LIN {X -167.693,Y -83.818,Z 210.000,A 0.000,B 0.000,C 180.000,E1 0.000} C_DIS
LIN {X -163.156,Y -92.341,Z 210.000,A 0.000,B 0.000,C 180.000,E1 0.000} C_DIS
LIN {X -158.186,Y -100.617,Z 210.000,A 0.000,B 0.000,C 180.000,E1 0.000} C_DIS
LIN {X -152.797,Y -108.627,Z 210.000,A 0.000,B 0.000,C 180.000,E1 0.000} C_DIS
LIN {X -147.002,Y -116.348,Z 210.000,A 0.000,B 0.000,C 180.000,E1 0.000} C_DIS
LIN {X -140.817,Y -123.762,Z 210.000,A 0.000,B 0.000,C 180.000,E1 0.000} C_DIS
LIN {X -134.260,Y -130.847,Z 210.000,A 0.000,B 0.000,C 180.000,E1 0.000} C_DIS
LIN {X -127.346,Y -137.585,Z 210.000,A 0.000,B 0.000,C 180.000,E1 0.000} C_DIS
LIN {X -120.095,Y -143.957,Z 210.000,A 0.000,B 0.000,C 180.000,E1 0.000} C_DIS
LIN {X -112.524,Y -149.949,Z 210.000,A 0.000,B 0.000,C 180.000,E1 0.000} C_DIS
LIN {X -104.656,Y -155.543,Z 210.000,A 0.000,B 0.000,C 180.000,E1 0.000} C_DIS
LIN {X -96.510,Y -160.725,Z 210.000,A 0.000,B 0.000,C 180.000,E1 0.000} C_DIS
LIN {X -88.108,Y -165.480,Z 210.000,A 0.000,B 0.000,C 180.000,E1 0.000} C_DIS
LIN {X -79.474,Y -169.796,Z 210.000,A 0.000,B 0.000,C 180.000,E1 0.000} C_DIS
LIN {X -70.624,Y -173.663,Z 210.000,A 0.000,B 0.000,C 180.000,E1 0.000} C_DIS
LIN {X -61.594,Y -177.067,Z 210.000,A 0.000,B 0.000,C 180.000,E1 0.000} C_DIS
LIN {X -52.397,Y -180.003,Z 210.000,A 0.000,B 0.000,C 180.000,E1 0.000} C_DIS
LIN {X -43.061,Y -182.462,Z 210.000,A 0.000,B 0.000,C 180.000,E1 0.000} C_DIS
LIN {X -33.610,Y -184.437,Z 210.000,A 0.000,B 0.000,C 180.000,E1 0.000} C_DIS
LIN {X -24.072,Y -185.923,Z 210.000,A 0.000,B 0.000,C 180.000,E1 0.000} C_DIS
LIN {X -14.469,Y -186.915,Z 210.000,A 0.000,B 0.000,C 180.000,E1 0.000} C_DIS
LIN {X -4.827,Y -187.412,Z 210.000,A 0.000,B 0.000,C 180.000,E1 0.000} C_DIS
LIN {X 4.827,Y -187.412,Z 210.000,A 0.000,B 0.000,C 180.000,E1 0.000} C_DIS
LIN {X 14.469,Y -186.915,Z 210.000,A 0.000,B 0.000,C 180.000,E1 0.000} C_DIS
LIN {X 24.072,Y -185.923,Z 210.000,A 0.000,B 0.000,C 180.000,E1 0.000} C_DIS
LIN {X 33.610,Y -184.437,Z 210.000,A 0.000,B 0.000,C 180.000,E1 0.000} C_DIS
LIN {X 43.061,Y -182.462,Z 210.000,A 0.000,B 0.000,C 180.000,E1 0.000} C_DIS
LIN {X 52.397,Y -180.003,Z 210.000,A 0.000,B 0.000,C 180.000,E1 0.000} C_DIS
LIN {X 61.593,Y -177.068,Z 210.000,A 0.000,B 0.000,C 180.000,E1 0.000} C_DIS
LIN {X 70.627,Y -173.662,Z 210.000,A 0.000,B 0.000,C 180.000,E1 0.000} C_DIS
LIN {X 79.474,Y -169.796,Z 210.000,A 0.000,B 0.000,C 180.000,E1 0.000} C_DIS
LIN {X 88.108,Y -165.480,Z 210.000,A 0.000,B 0.000,C 180.000,E1 0.000} C_DIS
LIN {X 96.510,Y -160.725,Z 210.000,A 0.000,B 0.000,C 180.000,E1 0.000} C_DIS
LIN {X 104.656,Y -155.543,Z 210.000,A 0.000,B 0.000,C 180.000,E1 0.000} C_DIS
LIN {X 112.524,Y -149.949,Z 210.000,A 0.000,B 0.000,C 180.000,E1 0.000} C_DIS
LIN {X 120.095,Y -143.957,Z 210.000,A 0.000,B 0.000,C 180.000,E1 0.000} C_DIS
LIN {X 127.346,Y -137.585,Z 210.000,A 0.000,B 0.000,C 180.000,E1 0.000} C_DIS
LIN {X 134.261,Y -130.846,Z 210.000,A 0.000,B 0.000,C 180.000,E1 0.000} C_DIS
LIN {X 140.817,Y -123.762,Z 210.000,A 0.000,B 0.000,C 180.000,E1 0.000} C_DIS
LIN {X 147.002,Y -116.348,Z 210.000,A 0.000,B 0.000,C 180.000,E1 0.000} C_DIS
LIN {X 152.797,Y -108.627,Z 210.000,A 0.000,B 0.000,C 180.000,E1 0.000} C_DIS
LIN {X 158.186,Y -100.617,Z 210.000,A 0.000,B 0.000,C 180.000,E1 0.000} C_DIS
LIN {X 163.156,Y -92.341,Z 210.000,A 0.000,B 0.000,C 180.000,E1 0.000} C_DIS
LIN {X 167.693,Y -83.818,Z 210.000,A 0.000,B 0.000,C 180.000,E1 0.000} C_DIS
LIN {X 171.786,Y -75.075,Z 210.000,A 0.000,B 0.000,C 180.000,E1 0.000} C_DIS
LIN {X 175.422,Y -66.133,Z 210.000,A 0.000,B 0.000,C 180.000,E1 0.000} C_DIS
LIN {X 178.595,Y -57.013,Z 210.000,A 0.000,B 0.000,C 180.000,E1 0.000} C_DIS
LIN {X 181.293,Y -47.744,Z 210.000,A 0.000,B 0.000,C 180.000,E1 0.000} C_DIS
LIN {X 183.511,Y -38.347,Z 210.000,A 0.000,B 0.000,C 180.000,E1 0.000} C_DIS
LIN {X 185.241,Y -28.852,Z 210.000,A 0.000,B 0.000,C 180.000,E1 0.000} C_DIS
LIN {X 186.480,Y -19.276,Z 210.000,A 0.000,B 0.000,C 180.000,E1 0.000} C_DIS
LIN {X 187.226,Y -9.650,Z 210.000,A 0.000,B 0.000,C 180.000,E1 0.000} C_DIS
LIN {X 187.474,Y 0.000,Z 210.000,A 0.000,B 0.000,C 180.000,E1 0.000} C_DIS
LIN {X 187.226,Y 9.650,Z 210.000,A 0.000,B 0.000,C 180.000,E1 0.000} C_DIS
LIN {X 186.480,Y 19.276,Z 210.000,A 0.000,B 0.000,C 180.000,E1 0.000} C_DIS
LIN {X 185.241,Y 28.852,Z 210.000,A 0.000,B 0.000,C 180.000,E1 0.000} C_DIS
LIN {X 183.511,Y 38.347,Z 210.000,A 0.000,B 0.000,C 180.000,E1 0.000} C_DIS
LIN {X 181.293,Y 47.744,Z 210.000,A 0.000,B 0.000,C 180.000,E1 0.000} C_DIS
LIN {X 178.595,Y 57.013,Z 210.000,A 0.000,B 0.000,C 180.000,E1 0.000} C_DIS
LIN {X 175.422,Y 66.133,Z 210.000,A 0.000,B 0.000,C 180.000,E1 0.000} C_DIS
LIN {X 171.786,Y 75.075,Z 210.000,A 0.000,B 0.000,C 180.000,E1 0.000} C_DIS
LIN {X 167.693,Y 83.818,Z 210.000,A 0.000,B 0.000,C 180.000,E1 0.000} C_DIS
LIN {X 163.156,Y 92.341,Z 210.000,A 0.000,B 0.000,C 180.000,E1 0.000} C_DIS
LIN {X 158.186,Y 100.617,Z 210.000,A 0.000,B 0.000,C 180.000,E1 0.000} C_DIS
LIN {X 152.797,Y 108.627,Z 210.000,A 0.000,B 0.000,C 180.000,E1 0.000} C_DIS
LIN {X 147.002,Y 116.348,Z 210.000,A 0.000,B 0.000,C 180.000,E1 0.000} C_DIS
LIN {X 140.817,Y 123.762,Z 210.000,A 0.000,B 0.000,C 180.000,E1 0.000} C_DIS
LIN {X 134.260,Y 130.847,Z 210.000,A 0.000,B 0.000,C 180.000,E1 0.000} C_DIS
LIN {X 127.346,Y 137.585,Z 210.000,A 0.000,B 0.000,C 180.000,E1 0.000} C_DIS
LIN {X 120.095,Y 143.957,Z 210.000,A 0.000,B 0.000,C 180.000,E1 0.000} C_DIS
LIN {X 112.524,Y 149.949,Z 210.000,A 0.000,B 0.000,C 180.000,E1 0.000} C_DIS
LIN {X 104.656,Y 155.543,Z 210.000,A 0.000,B 0.000,C 180.000,E1 0.000} C_DIS
LIN {X 96.510,Y 160.725,Z 210.000,A 0.000,B 0.000,C 180.000,E1 0.000} C_DIS
LIN {X 88.108,Y 165.480,Z 210.000,A 0.000,B 0.000,C 180.000,E1 0.000} C_DIS
LIN {X 79.474,Y 169.796,Z 210.000,A 0.000,B 0.000,C 180.000,E1 0.000} C_DIS
LIN {X 70.624,Y 173.663,Z 210.000,A 0.000,B 0.000,C 180.000,E1 0.000} C_DIS
LIN {X 61.594,Y 177.067,Z 210.000,A 0.000,B 0.000,C 180.000,E1 0.000} C_DIS
LIN {X 52.397,Y 180.003,Z 210.000,A 0.000,B 0.000,C 180.000,E1 0.000} C_DIS
LIN {X 43.061,Y 182.462,Z 210.000,A 0.000,B 0.000,C 180.000,E1 0.000} C_DIS
LIN {X 33.610,Y 184.437,Z 210.000,A 0.000,B 0.000,C 180.000,E1 0.000} C_DIS
LIN {X 24.072,Y 185.923,Z 210.000,A 0.000,B 0.000,C 180.000,E1 0.000} C_DIS
LIN {X 14.469,Y 186.915,Z 210.000,A 0.000,B 0.000,C 180.000,E1 0.000} C_DIS
LIN {X 4.827,Y 187.412,Z 210.000,A 0.000,B 0.000,C 180.000,E1 0.000} C_DIS
LIN {X -4.827,Y 187.412,Z 210.000,A 0.000,B 0.000,C 180.000,E1 0.000} C_DIS
LIN {X -14.469,Y 186.915,Z 210.000,A 0.000,B 0.000,C 180.000,E1 0.000} C_DIS
LIN {X -24.072,Y 185.923,Z 210.000,A 0.000,B 0.000,C 180.000,E1 0.000} C_DIS
LIN {X -33.610,Y 184.437,Z 210.000,A 0.000,B 0.000,C 180.000,E1 0.000} C_DIS
LIN {X -43.061,Y 182.462,Z 210.000,A 0.000,B 0.000,C 180.000,E1 0.000} C_DIS
LIN {X -52.397,Y 180.003,Z 210.000,A 0.000,B 0.000,C 180.000,E1 0.000} C_DIS
LIN {X -61.593,Y 177.068,Z 210.000,A 0.000,B 0.000,C 180.000,E1 0.000} C_DIS
LIN {X -70.627,Y 173.662,Z 210.000,A 0.000,B 0.000,C 180.000,E1 0.000} C_DIS
LIN {X -79.474,Y 169.796,Z 210.000,A 0.000,B 0.000,C 180.000,E1 0.000} C_DIS
LIN {X -88.108,Y 165.480,Z 210.000,A 0.000,B 0.000,C 180.000,E1 0.000} C_DIS
LIN {X -96.510,Y 160.725,Z 210.000,A 0.000,B 0.000,C 180.000,E1 0.000} C_DIS
LIN {X -104.656,Y 155.543,Z 210.000,A 0.000,B 0.000,C 180.000,E1 0.000} C_DIS
LIN {X -112.524,Y 149.949,Z 210.000,A 0.000,B 0.000,C 180.000,E1 0.000} C_DIS
LIN {X -120.095,Y 143.957,Z 210.000,A 0.000,B 0.000,C 180.000,E1 0.000} C_DIS
LIN {X -127.346,Y 137.585,Z 210.000,A 0.000,B 0.000,C 180.000,E1 0.000} C_DIS
LIN {X -134.261,Y 130.846,Z 210.000,A 0.000,B 0.000,C 180.000,E1 0.000} C_DIS
LIN {X -140.817,Y 123.762,Z 210.000,A 0.000,B 0.000,C 180.000,E1 0.000} C_DIS
LIN {X -147.002,Y 116.348,Z 210.000,A 0.000,B 0.000,C 180.000,E1 0.000} C_DIS
LIN {X -152.797,Y 108.627,Z 210.000,A 0.000,B 0.000,C 180.000,E1 0.000} C_DIS
LIN {X -158.186,Y 100.617,Z 210.000,A 0.000,B 0.000,C 180.000,E1 0.000} C_DIS
LIN {X -163.156,Y 92.341,Z 210.000,A 0.000,B 0.000,C 180.000,E1 0.000} C_DIS
LIN {X -167.693,Y 83.818,Z 210.000,A 0.000,B 0.000,C 180.000,E1 0.000} C_DIS
LIN {X -171.786,Y 75.075,Z 210.000,A 0.000,B 0.000,C 180.000,E1 0.000} C_DIS
LIN {X -175.422,Y 66.133,Z 210.000,A 0.000,B 0.000,C 180.000,E1 0.000} C_DIS
LIN {X -178.595,Y 57.013,Z 210.000,A 0.000,B 0.000,C 180.000,E1 0.000} C_DIS
LIN {X -181.293,Y 47.744,Z 210.000,A 0.000,B 0.000,C 180.000,E1 0.000} C_DIS
LIN {X -183.511,Y 38.347,Z 210.000,A 0.000,B 0.000,C 180.000,E1 0.000} C_DIS
LIN {X -185.241,Y 28.852,Z 210.000,A 0.000,B 0.000,C 180.000,E1 0.000} C_DIS
LIN {X -186.480,Y 19.276,Z 210.000,A 0.000,B 0.000,C 180.000,E1 0.000} C_DIS
LIN {X -187.226,Y 9.650,Z 210.000,A 0.000,B 0.000,C 180.000,E1 0.000} C_DIS
LIN {X -187.474,Y 0.000,Z 210.000,A 0.000,B 0.000,C 180.000,E1 0.000} C_DIS
LIN {X -187.226,Y -9.650,Z 210.000,A 0.000,B 0.000,C 180.000,E1 0.000} C_DIS
LIN {X -186.480,Y -19.276,Z 210.000,A 0.000,B 0.000,C 180.000,E1 0.000} C_DIS
LIN {X -185.241,Y -28.852,Z 210.000,A 0.000,B 0.000,C 180.000,E1 0.000} C_DIS
LIN {X -183.511,Y -38.347,Z 210.000,A 0.000,B 0.000,C 180.000,E1 0.000} C_DIS
;rapid-leaky
$VEL.CP=0.3
LIN {X -168.490,Y -19.914,Z 210.000,A 0.000,B 0.000,C 180.000,E1 0.000} C_DIS
;bead-sparse_infill
$VEL.CP=0.48
LIN {X -19.905,Y -168.499,Z 210.000,A 0.000,B 0.000,C 180.000,E1 0.000} C_DIS
LIN {X -13.098,Y -169.202,Z 210.000,A 0.000,B 0.000,C 180.000,E1 0.000} C_DIS
LIN {X -4.370,Y -169.652,Z 210.000,A 0.000,B 0.000,C 180.000,E1 0.000} C_DIS
LIN {X 4.370,Y -169.652,Z 210.000,A 0.000,B 0.000,C 180.000,E1 0.000} C_DIS
LIN {X 13.098,Y -169.202,Z 210.000,A 0.000,B 0.000,C 180.000,E1 0.000} C_DIS
LIN {X 21.791,Y -168.304,Z 210.000,A 0.000,B 0.000,C 180.000,E1 0.000} C_DIS
LIN {X 30.424,Y -166.959,Z 210.000,A 0.000,B 0.000,C 180.000,E1 0.000} C_DIS
LIN {X 38.980,Y -165.171,Z 210.000,A 0.000,B 0.000,C 180.000,E1 0.000} C_DIS
LIN {X 47.432,Y -162.945,Z 210.000,A 0.000,B 0.000,C 180.000,E1 0.000} C_DIS
LIN {X 55.756,Y -160.288,Z 210.000,A 0.000,B 0.000,C 180.000,E1 0.000} C_DIS
LIN {X 63.934,Y -157.205,Z 210.000,A 0.000,B 0.000,C 180.000,E1 0.000} C_DIS
LIN {X 71.943,Y -153.705,Z 210.000,A 0.000,B 0.000,C 180.000,E1 0.000} C_DIS
LIN {X 79.759,Y -149.798,Z 210.000,A 0.000,B 0.000,C 180.000,E1 0.000} C_DIS
LIN {X 87.365,Y -145.494,Z 210.000,A 0.000,B 0.000,C 180.000,E1 0.000} C_DIS
LIN {X 94.738,Y -140.804,Z 210.000,A 0.000,B 0.000,C 180.000,E1 0.000} C_DIS
LIN {X 101.861,Y -135.739,Z 210.000,A 0.000,B 0.000,C 180.000,E1 0.000} C_DIS
LIN {X 103.230,Y -134.656,Z 210.000,A 0.000,B 0.000,C 180.000,E1 0.000} C_DIS
LIN {X -134.648,Y 103.222,Z 210.000,A 0.000,B 0.000,C 180.000,E1 0.000} C_DIS
LIN {X -133.072,Y 105.322,Z 210.000,A 0.000,B 0.000,C 180.000,E1 0.000} C_DIS
LIN {X -127.472,Y 112.034,Z 210.000,A 0.000,B 0.000,C 180.000,E1 0.000} C_DIS
LIN {X -121.538,Y 118.447,Z 210.000,A 0.000,B 0.000,C 180.000,E1 0.000} C_DIS
LIN {X -115.278,Y 124.547,Z 210.000,A 0.000,B 0.000,C 180.000,E1 0.000} C_DIS
LIN {X -108.715,Y 130.315,Z 210.000,A 0.000,B 0.000,C 180.000,E1 0.000} C_DIS
LIN {X -101.861,Y 135.739,Z 210.000,A 0.000,B 0.000,C 180.000,E1 0.000} C_DIS
LIN {X -94.738,Y 140.804,Z 210.000,A 0.000,B 0.000,C 180.000,E1 0.000} C_DIS
LIN {X -87.365,Y 145.494,Z 210.000,A 0.000,B 0.000,C 180.000,E1 0.000} C_DIS
LIN {X -79.759,Y 149.798,Z 210.000,A 0.000,B 0.000,C 180.000,E1 0.000} C_DIS
LIN {X -71.943,Y 153.705,Z 210.000,A 0.000,B 0.000,C 180.000,E1 0.000} C_DIS
LIN {X -63.934,Y 157.205,Z 210.000,A 0.000,B 0.000,C 180.000,E1 0.000} C_DIS
LIN {X -55.756,Y 160.288,Z 210.000,A 0.000,B 0.000,C 180.000,E1 0.000} C_DIS
LIN {X -47.432,Y 162.945,Z 210.000,A 0.000,B 0.000,C 180.000,E1 0.000} C_DIS
LIN {X -39.486,Y 165.038,Z 210.000,A 0.000,B 0.000,C 180.000,E1 0.000} C_DIS
LIN {X 165.002,Y -39.451,Z 210.000,A 0.000,B 0.000,C 180.000,E1 0.000} C_DIS
;rapid-leaky
$VEL.CP=0.3
LIN {X 123.449,Y 147.980,Z 220.000,A 0.000,B 0.000,C 180.000,E1 0.000} C_DIS
;bead-perimeter_outer
$VEL.CP=0.45
LIN {X 115.668,Y 154.139,Z 220.000,A 0.000,B 0.000,C 180.000,E1 0.000} C_DIS
LIN {X 107.580,Y 159.888,Z 220.000,A 0.000,B 0.000,C 180.000,E1 0.000} C_DIS
LIN {X 99.207,Y 165.214,Z 220.000,A 0.000,B 0.000,C 180.000,E1 0.000} C_DIS
LIN {X 90.570,Y 170.102,Z 220.000,A 0.000,B 0.000,C 180.000,E1 0.000} C_DIS
LIN {X 81.693,Y 174.539,Z 220.000,A 0.000,B 0.000,C 180.000,E1 0.000} C_DIS
LIN {X 72.600,Y 178.514,Z 220.000,A 0.000,B 0.000,C 180.000,E1 0.000} C_DIS
LIN {X 63.314,Y 182.015,Z 220.000,A 0.000,B 0.000,C 180.000,E1 0.000} C_DIS
LIN {X 53.861,Y 185.032,Z 220.000,A 0.000,B 0.000,C 180.000,E1 0.000} C_DIS
LIN {X 44.264,Y 187.559,Z 220.000,A 0.000,B 0.000,C 180.000,E1 0.000} C_DIS
LIN {X 34.550,Y 189.589,Z 220.000,A 0.000,B 0.000,C 180.000,E1 0.000} C_DIS
LIN {X 24.744,Y 191.116,Z 220.000,A 0.000,B 0.000,C 180.000,E1 0.000} C_DIS
LIN {X 14.872,Y 192.137,Z 220.000,A 0.000,B 0.000,C 180.000,E1 0.000} C_DIS
LIN {X 4.962,Y 192.648,Z 220.000,A 0.000,B 0.000,C 180.000,E1 0.000} C_DIS
LIN {X -4.962,Y 192.648,Z 220.000,A 0.000,B 0.000,C 180.000,E1 0.000} C_DIS
LIN {X -14.872,Y 192.137,Z 220.000,A 0.000,B 0.000,C 180.000,E1 0.000} C_DIS
LIN {X -24.744,Y 191.116,Z 220.000,A 0.000,B 0.000,C 180.000,E1 0.000} C_DIS
LIN {X -34.550,Y 189.589,Z 220.000,A 0.000,B 0.000,C 180.000,E1 0.000} C_DIS
LIN {X -44.264,Y 187.559,Z 220.000,A 0.000,B 0.000,C 180.000,E1 0.000} C_DIS
LIN {X -53.861,Y 185.032,Z 220.000,A 0.000,B 0.000,C 180.000,E1 0.000} C_DIS
LIN {X -63.314,Y 182.015,Z 220.000,A 0.000,B 0.000,C 180.000,E1 0.000} C_DIS
LIN {X -72.600,Y 178.514,Z 220.000,A 0.000,B 0.000,C 180.000,E1 0.000} C_DIS
LIN {X -81.693,Y 174.539,Z 220.000,A 0.000,B 0.000,C 180.000,E1 0.000} C_DIS
LIN {X -83.733,Y 173.520,Z 220.000,A 0.000,B 0.000,C 180.000,E1 0.000} C_DIS
LIN {X -90.570,Y 170.102,Z 220.000,A 0.000,B 0.000,C 180.000,E1 0.000} C_DIS
LIN {X -99.207,Y 165.214,Z 220.000,A 0.000,B 0.000,C 180.000,E1 0.000} C_DIS
LIN {X -107.580,Y 159.888,Z 220.000,A 0.000,B 0.000,C 180.000,E1 0.000} C_DIS
LIN {X -115.668,Y 154.139,Z 220.000,A 0.000,B 0.000,C 180.000,E1 0.000} C_DIS
LIN {X -123.449,Y 147.980,Z 220.000,A 0.000,B 0.000,C 180.000,E1 0.000} C_DIS
LIN {X -130.904,Y 141.428,Z 220.000,A 0.000,B 0.000,C 180.000,E1 0.000} C_DIS
LIN {X -138.011,Y 134.501,Z 220.000,A 0.000,B 0.000,C 180.000,E1 0.000} C_DIS
LIN {X -144.752,Y 127.219,Z 220.000,A 0.000,B 0.000,C 180.000,E1 0.000} C_DIS
LIN {X -151.109,Y 119.599,Z 220.000,A 0.000,B 0.000,C 180.000,E1 0.000} C_DIS
LIN {X -157.065,Y 111.662,Z 220.000,A 0.000,B 0.000,C 180.000,E1 0.000} C_DIS
LIN {X -162.605,Y 103.428,Z 220.000,A 0.000,B 0.000,C 180.000,E1 0.000} C_DIS
LIN {X -167.714,Y 94.920,Z 220.000,A 0.000,B 0.000,C 180.000,E1 0.000} C_DIS
LIN {X -172.378,Y 86.160,Z 220.000,A 0.000,B 0.000,C 180.000,E1 0.000} C_DIS
LIN {X -176.585,Y 77.173,Z 220.000,A 0.000,B 0.000,C 180.000,E1 0.000} C_DIS
LIN {X -180.323,Y 67.979,Z 220.000,A 0.000,B 0.000,C 180.000,E1 0.000} C_DIS
LIN {X -183.583,Y 58.607,Z 220.000,A 0.000,B 0.000,C 180.000,E1 0.000} C_DIS
LIN {X -186.358,Y 49.078,Z 220.000,A 0.000,B 0.000,C 180.000,E1 0.000} C_DIS
LIN {X -188.637,Y 39.420,Z 220.000,A 0.000,B 0.000,C 180.000,E1 0.000} C_DIS
LIN {X -190.416,Y 29.656,Z 220.000,A 0.000,B 0.000,C 180.000,E1 0.000} C_DIS
LIN {X -191.690,Y 19.814,Z 220.000,A 0.000,B 0.000,C 180.000,E1 0.000} C_DIS
LIN {X -192.456,Y 9.921,Z 220.000,A 0.000,B 0.000,C 180.000,E1 0.000} C_DIS
LIN {X -192.711,Y 0.000,Z 220.000,A 0.000,B 0.000,C 180.000,E1 0.000} C_DIS
LIN {X -192.456,Y -9.921,Z 220.000,A 0.000,B 0.000,C 180.000,E1 0.000} C_DIS
LIN {X -191.690,Y -19.814,Z 220.000,A 0.000,B 0.000,C 180.000,E1 0.000} C_DIS
LIN {X -190.416,Y -29.656,Z 220.000,A 0.000,B 0.000,C 180.000,E1 0.000} C_DIS
LIN {X -188.637,Y -39.420,Z 220.000,A 0.000,B 0.000,C 180.000,E1 0.000} C_DIS
LIN {X -186.358,Y -49.078,Z 220.000,A 0.000,B 0.000,C 180.000,E1 0.000} C_DIS
LIN {X -183.583,Y -58.607,Z 220.000,A 0.000,B 0.000,C 180.000,E1 0.000} C_DIS
LIN {X -180.323,Y -67.980,Z 220.000,A 0.000,B 0.000,C 180.000,E1 0.000} C_DIS
LIN {X -176.585,Y -77.173,Z 220.000,A 0.000,B 0.000,C 180.000,E1 0.000} C_DIS
LIN {X -172.378,Y -86.160,Z 220.000,A 0.000,B 0.000,C 180.000,E1 0.000} C_DIS
LIN {X -167.714,Y -94.920,Z 220.000,A 0.000,B 0.000,C 180.000,E1 0.000} C_DIS
LIN {X -162.605,Y -103.428,Z 220.000,A 0.000,B 0.000,C 180.000,E1 0.000} C_DIS
LIN {X -157.065,Y -111.662,Z 220.000,A 0.000,B 0.000,C 180.000,E1 0.000} C_DIS
LIN {X -151.109,Y -119.599,Z 220.000,A 0.000,B 0.000,C 180.000,E1 0.000} C_DIS
LIN {X -144.752,Y -127.219,Z 220.000,A 0.000,B 0.000,C 180.000,E1 0.000} C_DIS
LIN {X -138.011,Y -134.501,Z 220.000,A 0.000,B 0.000,C 180.000,E1 0.000} C_DIS
LIN {X -130.904,Y -141.428,Z 220.000,A 0.000,B 0.000,C 180.000,E1 0.000} C_DIS
LIN {X -123.449,Y -147.980,Z 220.000,A 0.000,B 0.000,C 180.000,E1 0.000} C_DIS
LIN {X -115.668,Y -154.139,Z 220.000,A 0.000,B 0.000,C 180.000,E1 0.000} C_DIS
LIN {X -107.580,Y -159.888,Z 220.000,A 0.000,B 0.000,C 180.000,E1 0.000} C_DIS
LIN {X -99.207,Y -165.214,Z 220.000,A 0.000,B 0.000,C 180.000,E1 0.000} C_DIS
LIN {X -90.570,Y -170.102,Z 220.000,A 0.000,B 0.000,C 180.000,E1 0.000} C_DIS
LIN {X -81.693,Y -174.539,Z 220.000,A 0.000,B 0.000,C 180.000,E1 0.000} C_DIS
LIN {X -72.600,Y -178.514,Z 220.000,A 0.000,B 0.000,C 180.000,E1 0.000} C_DIS
LIN {X -63.314,Y -182.015,Z 220.000,A 0.000,B 0.000,C 180.000,E1 0.000} C_DIS
LIN {X -53.861,Y -185.032,Z 220.000,A 0.000,B 0.000,C 180.000,E1 0.000} C_DIS
LIN {X -44.264,Y -187.559,Z 220.000,A 0.000,B 0.000,C 180.000,E1 0.000} C_DIS
LIN {X -34.550,Y -189.589,Z 220.000,A 0.000,B 0.000,C 180.000,E1 0.000} C_DIS
LIN {X -24.744,Y -191.116,Z 220.000,A 0.000,B 0.000,C 180.000,E1 0.000} C_DIS
LIN {X -14.872,Y -192.137,Z 220.000,A 0.000,B 0.000,C 180.000,E1 0.000} C_DIS
LIN {X -4.962,Y -192.648,Z 220.000,A 0.000,B 0.000,C 180.000,E1 0.000} C_DIS
LIN {X 4.962,Y -192.648,Z 220.000,A 0.000,B 0.000,C 180.000,E1 0.000} C_DIS
LIN {X 14.872,Y -192.137,Z 220.000,A 0.000,B 0.000,C 180.000,E1 0.000} C_DIS
LIN {X 24.744,Y -191.116,Z 220.000,A 0.000,B 0.000,C 180.000,E1 0.000} C_DIS
LIN {X 34.550,Y -189.589,Z 220.000,A 0.000,B 0.000,C 180.000,E1 0.000} C_DIS
LIN {X 44.264,Y -187.559,Z 220.000,A 0.000,B 0.000,C 180.000,E1 0.000} C_DIS
LIN {X 53.861,Y -185.032,Z 220.000,A 0.000,B 0.000,C 180.000,E1 0.000} C_DIS
LIN {X 63.314,Y -182.015,Z 220.000,A 0.000,B 0.000,C 180.000,E1 0.000} C_DIS
LIN {X 72.600,Y -178.514,Z 220.000,A 0.000,B 0.000,C 180.000,E1 0.000} C_DIS
LIN {X 81.693,Y -174.539,Z 220.000,A 0.000,B 0.000,C 180.000,E1 0.000} C_DIS
LIN {X 90.570,Y -170.102,Z 220.000,A 0.000,B 0.000,C 180.000,E1 0.000} C_DIS
LIN {X 99.207,Y -165.214,Z 220.000,A 0.000,B 0.000,C 180.000,E1 0.000} C_DIS
LIN {X 107.580,Y -159.888,Z 220.000,A 0.000,B 0.000,C 180.000,E1 0.000} C_DIS
LIN {X 115.668,Y -154.139,Z 220.000,A 0.000,B 0.000,C 180.000,E1 0.000} C_DIS
LIN {X 123.449,Y -147.980,Z 220.000,A 0.000,B 0.000,C 180.000,E1 0.000} C_DIS
LIN {X 130.904,Y -141.428,Z 220.000,A 0.000,B 0.000,C 180.000,E1 0.000} C_DIS
LIN {X 138.011,Y -134.501,Z 220.000,A 0.000,B 0.000,C 180.000,E1 0.000} C_DIS
LIN {X 144.752,Y -127.219,Z 220.000,A 0.000,B 0.000,C 180.000,E1 0.000} C_DIS
LIN {X 151.109,Y -119.599,Z 220.000,A 0.000,B 0.000,C 180.000,E1 0.000} C_DIS
LIN {X 157.065,Y -111.662,Z 220.000,A 0.000,B 0.000,C 180.000,E1 0.000} C_DIS
LIN {X 162.605,Y -103.428,Z 220.000,A 0.000,B 0.000,C 180.000,E1 0.000} C_DIS
LIN {X 167.714,Y -94.920,Z 220.000,A 0.000,B 0.000,C 180.000,E1 0.000} C_DIS
LIN {X 172.378,Y -86.160,Z 220.000,A 0.000,B 0.000,C 180.000,E1 0.000} C_DIS
LIN {X 176.585,Y -77.173,Z 220.000,A 0.000,B 0.000,C 180.000,E1 0.000} C_DIS
LIN {X 180.323,Y -67.979,Z 220.000,A 0.000,B 0.000,C 180.000,E1 0.000} C_DIS
LIN {X 183.583,Y -58.607,Z 220.000,A 0.000,B 0.000,C 180.000,E1 0.000} C_DIS
LIN {X 186.358,Y -49.078,Z 220.000,A 0.000,B 0.000,C 180.000,E1 0.000} C_DIS
LIN {X 188.637,Y -39.420,Z 220.000,A 0.000,B 0.000,C 180.000,E1 0.000} C_DIS
LIN {X 190.416,Y -29.656,Z 220.000,A 0.000,B 0.000,C 180.000,E1 0.000} C_DIS
LIN {X 191.690,Y -19.814,Z 220.000,A 0.000,B 0.000,C 180.000,E1 0.000} C_DIS
LIN {X 192.456,Y -9.921,Z 220.000,A 0.000,B 0.000,C 180.000,E1 0.000} C_DIS
LIN {X 192.711,Y 0.000,Z 220.000,A 0.000,B 0.000,C 180.000,E1 0.000} C_DIS
LIN {X 192.456,Y 9.921,Z 220.000,A 0.000,B 0.000,C 180.000,E1 0.000} C_DIS
LIN {X 191.690,Y 19.814,Z 220.000,A 0.000,B 0.000,C 180.000,E1 0.000} C_DIS
LIN {X 190.416,Y 29.656,Z 220.000,A 0.000,B 0.000,C 180.000,E1 0.000} C_DIS
LIN {X 188.637,Y 39.420,Z 220.000,A 0.000,B 0.000,C 180.000,E1 0.000} C_DIS
LIN {X 186.358,Y 49.078,Z 220.000,A 0.000,B 0.000,C 180.000,E1 0.000} C_DIS
LIN {X 183.583,Y 58.607,Z 220.000,A 0.000,B 0.000,C 180.000,E1 0.000} C_DIS
LIN {X 180.323,Y 67.980,Z 220.000,A 0.000,B 0.000,C 180.000,E1 0.000} C_DIS
LIN {X 176.585,Y 77.173,Z 220.000,A 0.000,B 0.000,C 180.000,E1 0.000} C_DIS
LIN {X 172.378,Y 86.160,Z 220.000,A 0.000,B 0.000,C 180.000,E1 0.000} C_DIS
LIN {X 167.714,Y 94.920,Z 220.000,A 0.000,B 0.000,C 180.000,E1 0.000} C_DIS
LIN {X 162.605,Y 103.428,Z 220.000,A 0.000,B 0.000,C 180.000,E1 0.000} C_DIS
LIN {X 157.065,Y 111.662,Z 220.000,A 0.000,B 0.000,C 180.000,E1 0.000} C_DIS
LIN {X 151.109,Y 119.599,Z 220.000,A 0.000,B 0.000,C 180.000,E1 0.000} C_DIS
LIN {X 144.752,Y 127.219,Z 220.000,A 0.000,B 0.000,C 180.000,E1 0.000} C_DIS
LIN {X 138.011,Y 134.501,Z 220.000,A 0.000,B 0.000,C 180.000,E1 0.000} C_DIS
LIN {X 130.904,Y 141.428,Z 220.000,A 0.000,B 0.000,C 180.000,E1 0.000} C_DIS
LIN {X 123.449,Y 147.980,Z 220.000,A 0.000,B 0.000,C 180.000,E1 0.000} C_DIS
;rapid-leaky
$VEL.CP=0.3
LIN {X 113.490,Y 136.044,Z 220.000,A 0.000,B 0.000,C 180.000,E1 0.000} C_DIS
;bead-perimeter_inner
$VEL.CP=0.45
LIN {X 106.338,Y 141.705,Z 220.000,A 0.000,B 0.000,C 180.000,E1 0.000} C_DIS
LIN {X 98.903,Y 146.990,Z 220.000,A 0.000,B 0.000,C 180.000,E1 0.000} C_DIS
LIN {X 91.204,Y 151.887,Z 220.000,A 0.000,B 0.000,C 180.000,E1 0.000} C_DIS
LIN {X 83.264,Y 156.381,Z 220.000,A 0.000,B 0.000,C 180.000,E1 0.000} C_DIS
LIN {X 75.103,Y 160.460,Z 220.000,A 0.000,B 0.000,C 180.000,E1 0.000} C_DIS
LIN {X 66.743,Y 164.114,Z 220.000,A 0.000,B 0.000,C 180.000,E1 0.000} C_DIS
LIN {X 58.207,Y 167.332,Z 220.000,A 0.000,B 0.000,C 180.000,E1 0.000} C_DIS
LIN {X 49.517,Y 170.106,Z 220.000,A 0.000,B 0.000,C 180.000,E1 0.000} C_DIS
LIN {X 40.693,Y 172.430,Z 220.000,A 0.000,B 0.000,C 180.000,E1 0.000} C_DIS
LIN {X 31.763,Y 174.296,Z 220.000,A 0.000,B 0.000,C 180.000,E1 0.000} C_DIS
LIN {X 22.748,Y 175.700,Z 220.000,A 0.000,B 0.000,C 180.000,E1 0.000} C_DIS
LIN {X 13.672,Y 176.639,Z 220.000,A 0.000,B 0.000,C 180.000,E1 0.000} C_DIS
LIN {X 4.562,Y 177.108,Z 220.000,A 0.000,B 0.000,C 180.000,E1 0.000} C_DIS
LIN {X -4.562,Y 177.108,Z 220.000,A 0.000,B 0.000,C 180.000,E1 0.000} C_DIS
LIN {X -13.672,Y 176.639,Z 220.000,A 0.000,B 0.000,C 180.000,E1 0.000} C_DIS
LIN {X -22.748,Y 175.700,Z 220.000,A 0.000,B 0.000,C 180.000,E1 0.000} C_DIS
LIN {X -31.763,Y 174.296,Z 220.000,A 0.000,B 0.000,C 180.000,E1 0.000} C_DIS
LIN {X -40.693,Y 172.430,Z 220.000,A 0.000,B 0.000,C 180.000,E1 0.000} C_DIS
LIN {X -49.517,Y 170.106,Z 220.000,A 0.000,B 0.000,C 180.000,E1 0.000} C_DIS
LIN {X -58.207,Y 167.332,Z 220.000,A 0.000,B 0.000,C 180.000,E1 0.000} C_DIS
LIN {X -66.743,Y 164.114,Z 220.000,A 0.000,B 0.000,C 180.000,E1 0.000} C_DIS
LIN {X -75.104,Y 160.460,Z 220.000,A 0.000,B 0.000,C 180.000,E1 0.000} C_DIS
LIN {X -76.785,Y 159.619,Z 220.000,A 0.000,B 0.000,C 180.000,E1 0.000} C_DIS
LIN {X -83.264,Y 156.381,Z 220.000,A 0.000,B 0.000,C 180.000,E1 0.000} C_DIS
LIN {X -91.204,Y 151.887,Z 220.000,A 0.000,B 0.000,C 180.000,E1 0.000} C_DIS
LIN {X -98.903,Y 146.990,Z 220.000,A 0.000,B 0.000,C 180.000,E1 0.000} C_DIS
LIN {X -106.338,Y 141.705,Z 220.000,A 0.000,B 0.000,C 180.000,E1 0.000} C_DIS
LIN {X -113.490,Y 136.044,Z 220.000,A 0.000,B 0.000,C 180.000,E1 0.000} C_DIS
LIN {X -120.344,Y 130.020,Z 220.000,A 0.000,B 0.000,C 180.000,E1 0.000} C_DIS
LIN {X -126.878,Y 123.652,Z 220.000,A 0.000,B 0.000,C 180.000,E1 0.000} C_DIS
LIN {X -133.076,Y 116.956,Z 220.000,A 0.000,B 0.000,C 180.000,E1 0.000} C_DIS
LIN {X -138.920,Y 109.951,Z 220.000,A 0.000,B 0.000,C 180.000,E1 0.000} C_DIS
LIN {X -144.395,Y 102.655,Z 220.000,A 0.000,B 0.000,C 180.000,E1 0.000} C_DIS
LIN {X -149.488,Y 95.085,Z 220.000,A 0.000,B 0.000,C 180.000,E1 0.000} C_DIS
LIN {X -154.185,Y 87.263,Z 220.000,A 0.000,B 0.000,C 180.000,E1 0.000} C_DIS
LIN {X -158.474,Y 79.209,Z 220.000,A 0.000,B 0.000,C 180.000,E1 0.000} C_DIS
LIN {X -162.341,Y 70.948,Z 220.000,A 0.000,B 0.000,C 180.000,E1 0.000} C_DIS
LIN {X -165.777,Y 62.496,Z 220.000,A 0.000,B 0.000,C 180.000,E1 0.000} C_DIS
LIN {X -168.775,Y 53.879,Z 220.000,A 0.000,B 0.000,C 180.000,E1 0.000} C_DIS
LIN {X -171.325,Y 45.118,Z 220.000,A 0.000,B 0.000,C 180.000,E1 0.000} C_DIS
LIN {X -173.421,Y 36.240,Z 220.000,A 0.000,B 0.000,C 180.000,E1 0.000} C_DIS
LIN {X -175.056,Y 27.264,Z 220.000,A 0.000,B 0.000,C 180.000,E1 0.000} C_DIS
LIN {X -176.227,Y 18.215,Z 220.000,A 0.000,B 0.000,C 180.000,E1 0.000} C_DIS
LIN {X -176.931,Y 9.120,Z 220.000,A 0.000,B 0.000,C 180.000,E1 0.000} C_DIS
LIN {X -177.166,Y 0.000,Z 220.000,A 0.000,B 0.000,C 180.000,E1 0.000} C_DIS
LIN {X -176.931,Y -9.120,Z 220.000,A 0.000,B 0.000,C 180.000,E1 0.000} C_DIS
LIN {X -176.227,Y -18.215,Z 220.000,A 0.000,B 0.000,C 180.000,E1 0.000} C_DIS
LIN {X -175.056,Y -27.264,Z 220.000,A 0.000,B 0.000,C 180.000,E1 0.000} C_DIS
LIN {X -173.420,Y -36.241,Z 220.000,A 0.000,B 0.000,C 180.000,E1 0.000} C_DIS
LIN {X -171.325,Y -45.118,Z 220.000,A 0.000,B 0.000,C 180.000,E1 0.000} C_DIS
LIN {X -168.775,Y -53.879,Z 220.000,A 0.000,B 0.000,C 180.000,E1 0.000} C_DIS
LIN {X -165.777,Y -62.497,Z 220.000,A 0.000,B 0.000,C 180.000,E1 0.000} C_DIS
LIN {X -162.341,Y -70.948,Z 220.000,A 0.000,B 0.000,C 180.000,E1 0.000} C_DIS
LIN {X -158.474,Y -79.209,Z 220.000,A 0.000,B 0.000,C 180.000,E1 0.000} C_DIS
LIN {X -154.185,Y -87.263,Z 220.000,A 0.000,B 0.000,C 180.000,E1 0.000} C_DIS
LIN {X -149.488,Y -95.085,Z 220.000,A 0.000,B 0.000,C 180.000,E1 0.000} C_DIS
LIN {X -144.395,Y -102.655,Z 220.000,A 0.000,B 0.000,C 180.000,E1 0.000} C_DIS
LIN {X -138.920,Y -109.951,Z 220.000,A 0.000,B 0.000,C 180.000,E1 0.000} C_DIS
LIN {X -133.076,Y -116.956,Z 220.000,A 0.000,B 0.000,C 180.000,E1 0.000} C_DIS
LIN {X -126.878,Y -123.652,Z 220.000,A 0.000,B 0.000,C 180.000,E1 0.000} C_DIS
LIN {X -120.344,Y -130.020,Z 220.000,A 0.000,B 0.000,C 180.000,E1 0.000} C_DIS
LIN {X -113.490,Y -136.044,Z 220.000,A 0.000,B 0.000,C 180.000,E1 0.000} C_DIS
LIN {X -106.338,Y -141.705,Z 220.000,A 0.000,B 0.000,C 180.000,E1 0.000} C_DIS
LIN {X -98.903,Y -146.990,Z 220.000,A 0.000,B 0.000,C 180.000,E1 0.000} C_DIS
LIN {X -91.204,Y -151.887,Z 220.000,A 0.000,B 0.000,C 180.000,E1 0.000} C_DIS
LIN {X -83.264,Y -156.381,Z 220.000,A 0.000,B 0.000,C 180.000,E1 0.000} C_DIS
LIN {X -75.103,Y -160.460,Z 220.000,A 0.000,B 0.000,C 180.000,E1 0.000} C_DIS
LIN {X -66.743,Y -164.114,Z 220.000,A 0.000,B 0.000,C 180.000,E1 0.000} C_DIS
LIN {X -58.207,Y -167.332,Z 220.000,A 0.000,B 0.000,C 180.000,E1 0.000} C_DIS
LIN {X -49.517,Y -170.106,Z 220.000,A 0.000,B 0.000,C 180.000,E1 0.000} C_DIS
LIN {X -40.693,Y -172.430,Z 220.000,A 0.000,B 0.000,C 180.000,E1 0.000} C_DIS
LIN {X -31.763,Y -174.296,Z 220.000,A 0.000,B 0.000,C 180.000,E1 0.000} C_DIS
LIN {X -22.748,Y -175.700,Z 220.000,A 0.000,B 0.000,C 180.000,E1 0.000} C_DIS
LIN {X -13.672,Y -176.639,Z 220.000,A 0.000,B 0.000,C 180.000,E1 0.000} C_DIS
LIN {X -4.562,Y -177.108,Z 220.000,A 0.000,B 0.000,C 180.000,E1 0.000} C_DIS
LIN {X 4.562,Y -177.108,Z 220.000,A 0.000,B 0.000,C 180.000,E1 0.000} C_DIS
LIN {X 13.672,Y -176.639,Z 220.000,A 0.000,B 0.000,C 180.000,E1 0.000} C_DIS
LIN {X 22.748,Y -175.700,Z 220.000,A 0.000,B 0.000,C 180.000,E1 0.000} C_DIS
LIN {X 31.763,Y -174.296,Z 220.000,A 0.000,B 0.000,C 180.000,E1 0.000} C_DIS
LIN {X 40.693,Y -172.430,Z 220.000,A 0.000,B 0.000,C 180.000,E1 0.000} C_DIS
LIN {X 49.517,Y -170.106,Z 220.000,A 0.000,B 0.000,C 180.000,E1 0.000} C_DIS
LIN {X 58.207,Y -167.332,Z 220.000,A 0.000,B 0.000,C 180.000,E1 0.000} C_DIS
LIN {X 66.743,Y -164.114,Z 220.000,A 0.000,B 0.000,C 180.000,E1 0.000} C_DIS
LIN {X 75.104,Y -160.460,Z 220.000,A 0.000,B 0.000,C 180.000,E1 0.000} C_DIS
LIN {X 83.264,Y -156.381,Z 220.000,A 0.000,B 0.000,C 180.000,E1 0.000} C_DIS
LIN {X 91.204,Y -151.887,Z 220.000,A 0.000,B 0.000,C 180.000,E1 0.000} C_DIS
LIN {X 98.903,Y -146.990,Z 220.000,A 0.000,B 0.000,C 180.000,E1 0.000} C_DIS
LIN {X 106.338,Y -141.705,Z 220.000,A 0.000,B 0.000,C 180.000,E1 0.000} C_DIS
LIN {X 113.490,Y -136.044,Z 220.000,A 0.000,B 0.000,C 180.000,E1 0.000} C_DIS
LIN {X 120.344,Y -130.020,Z 220.000,A 0.000,B 0.000,C 180.000,E1 0.000} C_DIS
LIN {X 126.878,Y -123.652,Z 220.000,A 0.000,B 0.000,C 180.000,E1 0.000} C_DIS
LIN {X 133.076,Y -116.956,Z 220.000,A 0.000,B 0.000,C 180.000,E1 0.000} C_DIS
LIN {X 138.920,Y -109.951,Z 220.000,A 0.000,B 0.000,C 180.000,E1 0.000} C_DIS
LIN {X 144.395,Y -102.655,Z 220.000,A 0.000,B 0.000,C 180.000,E1 0.000} C_DIS
LIN {X 149.488,Y -95.085,Z 220.000,A 0.000,B 0.000,C 180.000,E1 0.000} C_DIS
LIN {X 154.185,Y -87.263,Z 220.000,A 0.000,B 0.000,C 180.000,E1 0.000} C_DIS
LIN {X 158.474,Y -79.209,Z 220.000,A 0.000,B 0.000,C 180.000,E1 0.000} C_DIS
LIN {X 162.341,Y -70.948,Z 220.000,A 0.000,B 0.000,C 180.000,E1 0.000} C_DIS
LIN {X 165.777,Y -62.496,Z 220.000,A 0.000,B 0.000,C 180.000,E1 0.000} C_DIS
LIN {X 168.775,Y -53.879,Z 220.000,A 0.000,B 0.000,C 180.000,E1 0.000} C_DIS
LIN {X 171.325,Y -45.118,Z 220.000,A 0.000,B 0.000,C 180.000,E1 0.000} C_DIS
LIN {X 173.421,Y -36.240,Z 220.000,A 0.000,B 0.000,C 180.000,E1 0.000} C_DIS
LIN {X 175.056,Y -27.264,Z 220.000,A 0.000,B 0.000,C 180.000,E1 0.000} C_DIS
LIN {X 176.227,Y -18.215,Z 220.000,A 0.000,B 0.000,C 180.000,E1 0.000} C_DIS
LIN {X 176.931,Y -9.120,Z 220.000,A 0.000,B 0.000,C 180.000,E1 0.000} C_DIS
LIN {X 177.166,Y 0.000,Z 220.000,A 0.000,B 0.000,C 180.000,E1 0.000} C_DIS
LIN {X 176.931,Y 9.120,Z 220.000,A 0.000,B 0.000,C 180.000,E1 0.000} C_DIS
LIN {X 176.227,Y 18.215,Z 220.000,A 0.000,B 0.000,C 180.000,E1 0.000} C_DIS
LIN {X 175.056,Y 27.264,Z 220.000,A 0.000,B 0.000,C 180.000,E1 0.000} C_DIS
LIN {X 173.420,Y 36.241,Z 220.000,A 0.000,B 0.000,C 180.000,E1 0.000} C_DIS
LIN {X 171.325,Y 45.118,Z 220.000,A 0.000,B 0.000,C 180.000,E1 0.000} C_DIS
LIN {X 168.775,Y 53.879,Z 220.000,A 0.000,B 0.000,C 180.000,E1 0.000} C_DIS
LIN {X 165.777,Y 62.497,Z 220.000,A 0.000,B 0.000,C 180.000,E1 0.000} C_DIS
LIN {X 162.341,Y 70.948,Z 220.000,A 0.000,B 0.000,C 180.000,E1 0.000} C_DIS
LIN {X 158.474,Y 79.209,Z 220.000,A 0.000,B 0.000,C 180.000,E1 0.000} C_DIS
LIN {X 154.185,Y 87.263,Z 220.000,A 0.000,B 0.000,C 180.000,E1 0.000} C_DIS
LIN {X 149.488,Y 95.085,Z 220.000,A 0.000,B 0.000,C 180.000,E1 0.000} C_DIS
LIN {X 144.395,Y 102.655,Z 220.000,A 0.000,B 0.000,C 180.000,E1 0.000} C_DIS
LIN {X 138.920,Y 109.951,Z 220.000,A 0.000,B 0.000,C 180.000,E1 0.000} C_DIS
LIN {X 133.076,Y 116.956,Z 220.000,A 0.000,B 0.000,C 180.000,E1 0.000} C_DIS
LIN {X 126.878,Y 123.652,Z 220.000,A 0.000,B 0.000,C 180.000,E1 0.000} C_DIS
LIN {X 120.344,Y 130.020,Z 220.000,A 0.000,B 0.000,C 180.000,E1 0.000} C_DIS
LIN {X 113.490,Y 136.044,Z 220.000,A 0.000,B 0.000,C 180.000,E1 0.000} C_DIS
;rapid-leaky
$VEL.CP=0.3
LIN {X -32.380,Y 156.023,Z 220.000,A 0.000,B 0.000,C 180.000,E1 0.000} C_DIS
;bead-sparse_infill
$VEL.CP=0.45
LIN {X -156.082,Y 32.321,Z 220.000,A 0.000,B 0.000,C 180.000,E1 0.000} C_DIS
LIN {X -157.501,Y 24.531,Z 220.000,A 0.000,B 0.000,C 180.000,E1 0.000} C_DIS
LIN {X -158.556,Y 16.388,Z 220.000,A 0.000,B 0.000,C 180.000,E1 0.000} C_DIS
LIN {X -159.189,Y 8.206,Z 220.000,A 0.000,B 0.000,C 180.000,E1 0.000} C_DIS
LIN {X -159.400,Y 0.000,Z 220.000,A 0.000,B 0.000,C 180.000,E1 0.000} C_DIS
LIN {X -159.189,Y -8.206,Z 220.000,A 0.000,B 0.000,C 180.000,E1 0.000} C_DIS
LIN {X -158.556,Y -16.388,Z 220.000,A 0.000,B 0.000,C 180.000,E1 0.000} C_DIS
LIN {X -157.501,Y -24.531,Z 220.000,A 0.000,B 0.000,C 180.000,E1 0.000} C_DIS
LIN {X -156.030,Y -32.607,Z 220.000,A 0.000,B 0.000,C 180.000,E1 0.000} C_DIS
LIN {X -154.145,Y -40.593,Z 220.000,A 0.000,B 0.000,C 180.000,E1 0.000} C_DIS
LIN {X -151.850,Y -48.476,Z 220.000,A 0.000,B 0.000,C 180.000,E1 0.000} C_DIS
LIN {X -149.153,Y -56.231,Z 220.000,A 0.000,B 0.000,C 180.000,E1 0.000} C_DIS
LIN {X -146.062,Y -63.834,Z 220.000,A 0.000,B 0.000,C 180.000,E1 0.000} C_DIS
LIN {X -142.583,Y -71.265,Z 220.000,A 0.000,B 0.000,C 180.000,E1 0.000} C_DIS
LIN {X -138.724,Y -78.512,Z 220.000,A 0.000,B 0.000,C 180.000,E1 0.000} C_DIS
LIN {X -134.498,Y -85.550,Z 220.000,A 0.000,B 0.000,C 180.000,E1 0.000} C_DIS
LIN {X -129.915,Y -92.361,Z 220.000,A 0.000,B 0.000,C 180.000,E1 0.000} C_DIS
LIN {X -127.288,Y -95.862,Z 220.000,A 0.000,B 0.000,C 180.000,E1 0.000} C_DIS
LIN {X 95.895,Y 127.321,Z 220.000,A 0.000,B 0.000,C 180.000,E1 0.000} C_DIS
LIN {X 102.109,Y 122.402,Z 220.000,A 0.000,B 0.000,C 180.000,E1 0.000} C_DIS
LIN {X 108.276,Y 116.982,Z 220.000,A 0.000,B 0.000,C 180.000,E1 0.000} C_DIS
LIN {X 114.155,Y 111.252,Z 220.000,A 0.000,B 0.000,C 180.000,E1 0.000} C_DIS
LIN {X 119.732,Y 105.227,Z 220.000,A 0.000,B 0.000,C 180.000,E1 0.000} C_DIS
LIN {X 124.990,Y 98.926,Z 220.000,A 0.000,B 0.000,C 180.000,E1 0.000} C_DIS
LIN {X 129.915,Y 92.361,Z 220.000,A 0.000,B 0.000,C 180.000,E1 0.000} C_DIS
LIN {X 134.498,Y 85.550,Z 220.000,A 0.000,B 0.000,C 180.000,E1 0.000} C_DIS
LIN {X 138.724,Y 78.512,Z 220.000,A 0.000,B 0.000,C 180.000,E1 0.000} C_DIS
LIN {X 142.583,Y 71.265,Z 220.000,A 0.000,B 0.000,C 180.000,E1 0.000} C_DIS
LIN {X 146.062,Y 63.834,Z 220.000,A 0.000,B 0.000,C 180.000,E1 0.000} C_DIS
LIN {X 149.153,Y 56.231,Z 220.000,A 0.000,B 0.000,C 180.000,E1 0.000} C_DIS
LIN {X 151.850,Y 48.476,Z 220.000,A 0.000,B 0.000,C 180.000,E1 0.000} C_DIS
LIN {X 154.145,Y 40.593,Z 220.000,A 0.000,B 0.000,C 180.000,E1 0.000} C_DIS
LIN {X 156.030,Y 32.607,Z 220.000,A 0.000,B 0.000,C 180.000,E1 0.000} C_DIS
LIN {X 156.358,Y 30.806,Z 220.000,A 0.000,B 0.000,C 180.000,E1 0.000} C_DIS
LIN {X -30.801,Y -156.353,Z 220.000,A 0.000,B 0.000,C 180.000,E1 0.000} C_DIS
;rapid-leaky
$VEL.CP=0.3
LIN {X 181.123,Y 9.336,Z 230.000,A 0.000,B 0.000,C 180.000,E1 0.000} C_DIS
;bead-perimeter_outer
$VEL.CP=0.41
LIN {X 180.402,Y 18.647,Z 230.000,A 0.000,B 0.000,C 180.000,E1 0.000} C_DIS
LIN {X 179.203,Y 27.910,Z 230.000,A 0.000,B 0.000,C 180.000,E1 0.000} C_DIS
LIN {X 177.528,Y 37.099,Z 230.000,A 0.000,B 0.000,C 180.000,E1 0.000} C_DIS
LIN {X 175.383,Y 46.188,Z 230.000,A 0.000,B 0.000,C 180.000,E1 0.000} C_DIS
LIN {X 172.772,Y 55.155,Z 230.000,A 0.000,B 0.000,C 180.000,E1 0.000} C_DIS
LIN {X 169.704,Y 63.976,Z 230.000,A 0.000,B 0.000,C 180.000,E1 0.000} C_DIS
LIN {X 166.185,Y 72.628,Z 230.000,A 0.000,B 0.000,C 180.000,E1 0.000} C_DIS
LIN {X 162.227,Y 81.087,Z 230.000,A 0.000,B 0.000,C 180.000,E1 0.000} C_DIS
LIN {X 157.838,Y 89.330,Z 230.000,A 0.000,B 0.000,C 180.000,E1 0.000} C_DIS
LIN {X 156.768,Y 91.112,Z 230.000,A 0.000,B 0.000,C 180.000,E1 0.000} C_DIS
LIN {X 153.030,Y 97.337,Z 230.000,A 0.000,B 0.000,C 180.000,E1 0.000} C_DIS
LIN {X 147.816,Y 105.086,Z 230.000,A 0.000,B 0.000,C 180.000,E1 0.000} C_DIS
LIN {X 142.211,Y 112.556,Z 230.000,A 0.000,B 0.000,C 180.000,E1 0.000} C_DIS
LIN {X 136.228,Y 119.727,Z 230.000,A 0.000,B 0.000,C 180.000,E1 0.000} C_DIS
LIN {X 129.884,Y 126.582,Z 230.000,A 0.000,B 0.000,C 180.000,E1 0.000} C_DIS
LIN {X 123.196,Y 133.100,Z 230.000,A 0.000,B 0.000,C 180.000,E1 0.000} C_DIS
LIN {X 116.180,Y 139.266,Z 230.000,A 0.000,B 0.000,C 180.000,E1 0.000} C_DIS
LIN {X 108.856,Y 145.062,Z 230.000,A 0.000,B 0.000,C 180.000,E1 0.000} C_DIS
LIN {X 101.245,Y 150.473,Z 230.000,A 0.000,B 0.000,C 180.000,E1 0.000} C_DIS
LIN {X 93.365,Y 155.484,Z 230.000,A 0.000,B 0.000,C 180.000,E1 0.000} C_DIS
LIN {X 85.236,Y 160.085,Z 230.000,A 0.000,B 0.000,C 180.000,E1 0.000} C_DIS
LIN {X 76.883,Y 164.262,Z 230.000,A 0.000,B 0.000,C 180.000,E1 0.000} C_DIS
LIN {X 68.326,Y 168.001,Z 230.000,A 0.000,B 0.000,C 180.000,E1 0.000} C_DIS
LIN {X 59.586,Y 171.295,Z 230.000,A 0.000,B 0.000,C 180.000,E1 0.000} C_DIS
LIN {X 50.688,Y 174.136,Z 230.000,A 0.000,B 0.000,C 180.000,E1 0.000} C_DIS
LIN {X 41.657,Y 176.514,Z 230.000,A 0.000,B 0.000,C 180.000,E1 0.000} C_DIS
LIN {X 32.515,Y 178.425,Z 230.000,A 0.000,B 0.000,C 180.000,E1 0.000} C_DIS
LIN {X 23.287,Y 179.862,Z 230.000,A 0.000,B 0.000,C 180.000,E1 0.000} C_DIS
LIN {X 13.997,Y 180.822,Z 230.000,A 0.000,B 0.000,C 180.000,E1 0.000} C_DIS
LIN {X 4.669,Y 181.303,Z 230.000,A 0.000,B 0.000,C 180.000,E1 0.000} C_DIS
LIN {X -4.669,Y 181.303,Z 230.000,A 0.000,B 0.000,C 180.000,E1 0.000} C_DIS
LIN {X -13.997,Y 180.822,Z 230.000,A 0.000,B 0.000,C 180.000,E1 0.000} C_DIS
LIN {X -23.287,Y 179.862,Z 230.000,A 0.000,B 0.000,C 180.000,E1 0.000} C_DIS
LIN {X -32.515,Y 178.425,Z 230.000,A 0.000,B 0.000,C 180.000,E1 0.000} C_DIS
LIN {X -41.657,Y 176.514,Z 230.000,A 0.000,B 0.000,C 180.000,E1 0.000} C_DIS
LIN {X -50.688,Y 174.136,Z 230.000,A 0.000,B 0.000,C 180.000,E1 0.000} C_DIS
LIN {X -59.586,Y 171.295,Z 230.000,A 0.000,B 0.000,C 180.000,E1 0.000} C_DIS
LIN {X -68.326,Y 168.001,Z 230.000,A 0.000,B 0.000,C 180.000,E1 0.000} C_DIS
LIN {X -76.883,Y 164.262,Z 230.000,A 0.000,B 0.000,C 180.000,E1 0.000} C_DIS
LIN {X -85.236,Y 160.085,Z 230.000,A 0.000,B 0.000,C 180.000,E1 0.000} C_DIS
LIN {X -93.365,Y 155.484,Z 230.000,A 0.000,B 0.000,C 180.000,E1 0.000} C_DIS
LIN {X -101.245,Y 150.473,Z 230.000,A 0.000,B 0.000,C 180.000,E1 0.000} C_DIS
LIN {X -108.856,Y 145.062,Z 230.000,A 0.000,B 0.000,C 180.000,E1 0.000} C_DIS
LIN {X -116.180,Y 139.266,Z 230.000,A 0.000,B 0.000,C 180.000,E1 0.000} C_DIS
LIN {X -123.196,Y 133.100,Z 230.000,A 0.000,B 0.000,C 180.000,E1 0.000} C_DIS
LIN {X -129.884,Y 126.582,Z 230.000,A 0.000,B 0.000,C 180.000,E1 0.000} C_DIS
LIN {X -136.228,Y 119.727,Z 230.000,A 0.000,B 0.000,C 180.000,E1 0.000} C_DIS
LIN {X -142.211,Y 112.556,Z 230.000,A 0.000,B 0.000,C 180.000,E1 0.000} C_DIS
LIN {X -147.816,Y 105.086,Z 230.000,A 0.000,B 0.000,C 180.000,E1 0.000} C_DIS
LIN {X -153.030,Y 97.337,Z 230.000,A 0.000,B 0.000,C 180.000,E1 0.000} C_DIS
LIN {X -157.838,Y 89.330,Z 230.000,A 0.000,B 0.000,C 180.000,E1 0.000} C_DIS
LIN {X -162.227,Y 81.087,Z 230.000,A 0.000,B 0.000,C 180.000,E1 0.000} C_DIS
LIN {X -166.185,Y 72.628,Z 230.000,A 0.000,B 0.000,C 180.000,E1 0.000} C_DIS
LIN {X -169.704,Y 63.976,Z 230.000,A 0.000,B 0.000,C 180.000,E1 0.000} C_DIS
LIN {X -170.388,Y 62.012,Z 230.000,A 0.000,B 0.000,C 180.000,E1 0.000} C_DIS
LIN {X -172.772,Y 55.155,Z 230.000,A 0.000,B 0.000,C 180.000,E1 0.000} C_DIS
LIN {X -175.383,Y 46.188,Z 230.000,A 0.000,B 0.000,C 180.000,E1 0.000} C_DIS
LIN {X -177.528,Y 37.099,Z 230.000,A 0.000,B 0.000,C 180.000,E1 0.000} C_DIS
LIN {X -179.203,Y 27.910,Z 230.000,A 0.000,B 0.000,C 180.000,E1 0.000} C_DIS
LIN {X -180.402,Y 18.647,Z 230.000,A 0.000,B 0.000,C 180.000,E1 0.000} C_DIS
LIN {X -181.123,Y 9.336,Z 230.000,A 0.000,B 0.000,C 180.000,E1 0.000} C_DIS
LIN {X -181.363,Y 0.000,Z 230.000,A 0.000,B 0.000,C 180.000,E1 0.000} C_DIS
LIN {X -181.123,Y -9.336,Z 230.000,A 0.000,B 0.000,C 180.000,E1 0.000} C_DIS
LIN {X -180.402,Y -18.647,Z 230.000,A 0.000,B 0.000,C 180.000,E1 0.000} C_DIS
LIN {X -179.203,Y -27.910,Z 230.000,A 0.000,B 0.000,C 180.000,E1 0.000} C_DIS
LIN {X -177.528,Y -37.099,Z 230.000,A 0.000,B 0.000,C 180.000,E1 0.000} C_DIS
LIN {X -175.383,Y -46.188,Z 230.000,A 0.000,B 0.000,C 180.000,E1 0.000} C_DIS
LIN {X -172.772,Y -55.155,Z 230.000,A 0.000,B 0.000,C 180.000,E1 0.000} C_DIS
LIN {X -169.704,Y -63.976,Z 230.000,A 0.000,B 0.000,C 180.000,E1 0.000} C_DIS
LIN {X -166.185,Y -72.628,Z 230.000,A 0.000,B 0.000,C 180.000,E1 0.000} C_DIS
LIN {X -162.227,Y -81.087,Z 230.000,A 0.000,B 0.000,C 180.000,E1 0.000} C_DIS
LIN {X -157.838,Y -89.330,Z 230.000,A 0.000,B 0.000,C 180.000,E1 0.000} C_DIS
LIN {X -153.030,Y -97.337,Z 230.000,A 0.000,B 0.000,C 180.000,E1 0.000} C_DIS
LIN {X -147.816,Y -105.086,Z 230.000,A 0.000,B 0.000,C 180.000,E1 0.000} C_DIS
LIN {X -142.211,Y -112.556,Z 230.000,A 0.000,B 0.000,C 180.000,E1 0.000} C_DIS
LIN {X -136.228,Y -119.727,Z 230.000,A 0.000,B 0.000,C 180.000,E1 0.000} C_DIS
LIN {X -129.884,Y -126.582,Z 230.000,A 0.000,B 0.000,C 180.000,E1 0.000} C_DIS
LIN {X -123.196,Y -133.100,Z 230.000,A 0.000,B 0.000,C 180.000,E1 0.000} C_DIS
LIN {X -116.180,Y -139.266,Z 230.000,A 0.000,B 0.000,C 180.000,E1 0.000} C_DIS
LIN {X -108.856,Y -145.062,Z 230.000,A 0.000,B 0.000,C 180.000,E1 0.000} C_DIS
LIN {X -101.245,Y -150.473,Z 230.000,A 0.000,B 0.000,C 180.000,E1 0.000} C_DIS
LIN {X -93.365,Y -155.484,Z 230.000,A 0.000,B 0.000,C 180.000,E1 0.000} C_DIS
LIN {X -85.236,Y -160.085,Z 230.000,A 0.000,B 0.000,C 180.000,E1 0.000} C_DIS
LIN {X -76.883,Y -164.262,Z 230.000,A 0.000,B 0.000,C 180.000,E1 0.000} C_DIS
LIN {X -68.326,Y -168.001,Z 230.000,A 0.000,B 0.000,C 180.000,E1 0.000} C_DIS
LIN {X -59.586,Y -171.295,Z 230.000,A 0.000,B 0.000,C 180.000,E1 0.000} C_DIS
LIN {X -50.688,Y -174.136,Z 230.000,A 0.000,B 0.000,C 180.000,E1 0.000} C_DIS
LIN {X -41.657,Y -176.514,Z 230.000,A 0.000,B 0.000,C 180.000,E1 0.000} C_DIS
LIN {X -32.515,Y -178.425,Z 230.000,A 0.000,B 0.000,C 180.000,E1 0.000} C_DIS
LIN {X -23.287,Y -179.862,Z 230.000,A 0.000,B 0.000,C 180.000,E1 0.000} C_DIS
LIN {X -13.997,Y -180.822,Z 230.000,A 0.000,B 0.000,C 180.000,E1 0.000} C_DIS
LIN {X -4.669,Y -181.303,Z 230.000,A 0.000,B 0.000,C 180.000,E1 0.000} C_DIS
LIN {X 4.669,Y -181.303,Z 230.000,A 0.000,B 0.000,C 180.000,E1 0.000} C_DIS
LIN {X 13.997,Y -180.822,Z 230.000,A 0.000,B 0.000,C 180.000,E1 0.000} C_DIS
LIN {X 23.287,Y -179.862,Z 230.000,A 0.000,B 0.000,C 180.000,E1 0.000} C_DIS
LIN {X 32.515,Y -178.425,Z 230.000,A 0.000,B 0.000,C 180.000,E1 0.000} C_DIS
LIN {X 41.657,Y -176.514,Z 230.000,A 0.000,B 0.000,C 180.000,E1 0.000} C_DIS
LIN {X 50.688,Y -174.136,Z 230.000,A 0.000,B 0.000,C 180.000,E1 0.000} C_DIS
LIN {X 59.586,Y -171.295,Z 230.000,A 0.000,B 0.000,C 180.000,E1 0.000} C_DIS
LIN {X 68.326,Y -168.001,Z 230.000,A 0.000,B 0.000,C 180.000,E1 0.000} C_DIS
LIN {X 76.883,Y -164.262,Z 230.000,A 0.000,B 0.000,C 180.000,E1 0.000} C_DIS
LIN {X 85.236,Y -160.085,Z 230.000,A 0.000,B 0.000,C 180.000,E1 0.000} C_DIS
LIN {X 93.365,Y -155.484,Z 230.000,A 0.000,B 0.000,C 180.000,E1 0.000} C_DIS
LIN {X 101.245,Y -150.473,Z 230.000,A 0.000,B 0.000,C 180.000,E1 0.000} C_DIS
LIN {X 108.856,Y -145.062,Z 230.000,A 0.000,B 0.000,C 180.000,E1 0.000} C_DIS
LIN {X 116.180,Y -139.266,Z 230.000,A 0.000,B 0.000,C 180.000,E1 0.000} C_DIS
LIN {X 123.196,Y -133.100,Z 230.000,A 0.000,B 0.000,C 180.000,E1 0.000} C_DIS
LIN {X 129.884,Y -126.582,Z 230.000,A 0.000,B 0.000,C 180.000,E1 0.000} C_DIS
LIN {X 136.228,Y -119.727,Z 230.000,A 0.000,B 0.000,C 180.000,E1 0.000} C_DIS
LIN {X 142.211,Y -112.556,Z 230.000,A 0.000,B 0.000,C 180.000,E1 0.000} C_DIS
LIN {X 147.816,Y -105.086,Z 230.000,A 0.000,B 0.000,C 180.000,E1 0.000} C_DIS
LIN {X 153.030,Y -97.337,Z 230.000,A 0.000,B 0.000,C 180.000,E1 0.000} C_DIS
LIN {X 157.838,Y -89.330,Z 230.000,A 0.000,B 0.000,C 180.000,E1 0.000} C_DIS
LIN {X 162.227,Y -81.087,Z 230.000,A 0.000,B 0.000,C 180.000,E1 0.000} C_DIS
LIN {X 166.185,Y -72.628,Z 230.000,A 0.000,B 0.000,C 180.000,E1 0.000} C_DIS
LIN {X 169.704,Y -63.976,Z 230.000,A 0.000,B 0.000,C 180.000,E1 0.000} C_DIS
LIN {X 172.772,Y -55.155,Z 230.000,A 0.000,B 0.000,C 180.000,E1 0.000} C_DIS
LIN {X 175.383,Y -46.188,Z 230.000,A 0.000,B 0.000,C 180.000,E1 0.000} C_DIS
LIN {X 177.528,Y -37.099,Z 230.000,A 0.000,B 0.000,C 180.000,E1 0.000} C_DIS
LIN {X 179.203,Y -27.910,Z 230.000,A 0.000,B 0.000,C 180.000,E1 0.000} C_DIS
LIN {X 180.402,Y -18.647,Z 230.000,A 0.000,B 0.000,C 180.000,E1 0.000} C_DIS
LIN {X 181.123,Y -9.336,Z 230.000,A 0.000,B 0.000,C 180.000,E1 0.000} C_DIS
LIN {X 181.363,Y 0.000,Z 230.000,A 0.000,B 0.000,C 180.000,E1 0.000} C_DIS
LIN {X 181.123,Y 9.336,Z 230.000,A 0.000,B 0.000,C 180.000,E1 0.000} C_DIS
;rapid-leaky
$VEL.CP=0.3
LIN {X 165.598,Y 8.536,Z 230.000,A 0.000,B 0.000,C 180.000,E1 0.000} C_DIS
;bead-perimeter_inner
$VEL.CP=0.41
LIN {X 164.939,Y 17.048,Z 230.000,A 0.000,B 0.000,C 180.000,E1 0.000} C_DIS
LIN {X 163.843,Y 25.518,Z 230.000,A 0.000,B 0.000,C 180.000,E1 0.000} C_DIS
LIN {X 162.312,Y 33.919,Z 230.000,A 0.000,B 0.000,C 180.000,E1 0.000} C_DIS
LIN {X 160.351,Y 42.229,Z 230.000,A 0.000,B 0.000,C 180.000,E1 0.000} C_DIS
LIN {X 157.964,Y 50.427,Z 230.000,A 0.000,B 0.000,C 180.000,E1 0.000} C_DIS
LIN {X 155.158,Y 58.493,Z 230.000,A 0.000,B 0.000,C 180.000,E1 0.000} C_DIS
LIN {X 151.941,Y 66.403,Z 230.000,A 0.000,B 0.000,C 180.000,E1 0.000} C_DIS
LIN {X 148.322,Y 74.137,Z 230.000,A 0.000,B 0.000,C 180.000,E1 0.000} C_DIS
LIN {X 144.309,Y 81.674,Z 230.000,A 0.000,B 0.000,C 180.000,E1 0.000} C_DIS
LIN {X 143.445,Y 83.112,Z 230.000,A 0.000,B 0.000,C 180.000,E1 0.000} C_DIS
LIN {X 139.913,Y 88.994,Z 230.000,A 0.000,B 0.000,C 180.000,E1 0.000} C_DIS
LIN {X 135.146,Y 96.079,Z 230.000,A 0.000,B 0.000,C 180.000,E1 0.000} C_DIS
LIN {X 130.022,Y 102.908,Z 230.000,A 0.000,B 0.000,C 180.000,E1 0.000} C_DIS
LIN {X 124.551,Y 109.465,Z 230.000,A 0.000,B 0.000,C 180.000,E1 0.000} C_DIS
LIN {X 118.751,Y 115.732,Z 230.000,A 0.000,B 0.000,C 180.000,E1 0.000} C_DIS
LIN {X 112.636,Y 121.692,Z 230.000,A 0.000,B 0.000,C 180.000,E1 0.000} C_DIS
LIN {X 106.222,Y 127.329,Z 230.000,A 0.000,B 0.000,C 180.000,E1 0.000} C_DIS
LIN {X 99.526,Y 132.628,Z 230.000,A 0.000,B 0.000,C 180.000,E1 0.000} C_DIS
LIN {X 92.567,Y 137.576,Z 230.000,A 0.000,B 0.000,C 180.000,E1 0.000} C_DIS
LIN {X 85.363,Y 142.157,Z 230.000,A 0.000,B 0.000,C 180.000,E1 0.000} C_DIS
LIN {X 77.930,Y 146.364,Z 230.000,A 0.000,B 0.000,C 180.000,E1 0.000} C_DIS
LIN {X 70.292,Y 150.183,Z 230.000,A 0.000,B 0.000,C 180.000,E1 0.000} C_DIS
LIN {X 62.470,Y 153.601,Z 230.000,A 0.000,B 0.000,C 180.000,E1 0.000} C_DIS
LIN {X 54.479,Y 156.612,Z 230.000,A 0.000,B 0.000,C 180.000,E1 0.000} C_DIS
LIN {X 46.343,Y 159.210,Z 230.000,A 0.000,B 0.000,C 180.000,E1 0.000} C_DIS
LIN {X 38.086,Y 161.385,Z 230.000,A 0.000,B 0.000,C 180.000,E1 0.000} C_DIS
LIN {X 29.728,Y 163.132,Z 230.000,A 0.000,B 0.000,C 180.000,E1 0.000} C_DIS
LIN {X 21.292,Y 164.446,Z 230.000,A 0.000,B 0.000,C 180.000,E1 0.000} C_DIS
LIN {X 12.798,Y 165.324,Z 230.000,A 0.000,B 0.000,C 180.000,E1 0.000} C_DIS
LIN {X 4.269,Y 165.763,Z 230.000,A 0.000,B 0.000,C 180.000,E1 0.000} C_DIS
LIN {X -4.269,Y 165.763,Z 230.000,A 0.000,B 0.000,C 180.000,E1 0.000} C_DIS
LIN {X -12.798,Y 165.324,Z 230.000,A 0.000,B 0.000,C 180.000,E1 0.000} C_DIS
LIN {X -21.292,Y 164.446,Z 230.000,A 0.000,B 0.000,C 180.000,E1 0.000} C_DIS
LIN {X -29.728,Y 163.132,Z 230.000,A 0.000,B 0.000,C 180.000,E1 0.000} C_DIS
LIN {X -38.087,Y 161.385,Z 230.000,A 0.000,B 0.000,C 180.000,E1 0.000} C_DIS
LIN {X -46.343,Y 159.210,Z 230.000,A 0.000,B 0.000,C 180.000,E1 0.000} C_DIS
LIN {X -54.479,Y 156.612,Z 230.000,A 0.000,B 0.000,C 180.000,E1 0.000} C_DIS
LIN {X -62.470,Y 153.601,Z 230.000,A 0.000,B 0.000,C 180.000,E1 0.000} C_DIS
LIN {X -70.292,Y 150.183,Z 230.000,A 0.000,B 0.000,C 180.000,E1 0.000} C_DIS
LIN {X -77.930,Y 146.364,Z 230.000,A 0.000,B 0.000,C 180.000,E1 0.000} C_DIS
LIN {X -85.363,Y 142.157,Z 230.000,A 0.000,B 0.000,C 180.000,E1 0.000} C_DIS
LIN {X -92.567,Y 137.576,Z 230.000,A 0.000,B 0.000,C 180.000,E1 0.000} C_DIS
LIN {X -99.526,Y 132.628,Z 230.000,A 0.000,B 0.000,C 180.000,E1 0.000} C_DIS
LIN {X -106.222,Y 127.329,Z 230.000,A 0.000,B 0.000,C 180.000,E1 0.000} C_DIS
LIN {X -112.636,Y 121.692,Z 230.000,A 0.000,B 0.000,C 180.000,E1 0.000} C_DIS
LIN {X -118.751,Y 115.732,Z 230.000,A 0.000,B 0.000,C 180.000,E1 0.000} C_DIS
LIN {X -124.551,Y 109.465,Z 230.000,A 0.000,B 0.000,C 180.000,E1 0.000} C_DIS
LIN {X -130.022,Y 102.908,Z 230.000,A 0.000,B 0.000,C 180.000,E1 0.000} C_DIS
LIN {X -135.146,Y 96.079,Z 230.000,A 0.000,B 0.000,C 180.000,E1 0.000} C_DIS
LIN {X -139.913,Y 88.994,Z 230.000,A 0.000,B 0.000,C 180.000,E1 0.000} C_DIS
LIN {X -144.309,Y 81.673,Z 230.000,A 0.000,B 0.000,C 180.000,E1 0.000} C_DIS
LIN {X -148.322,Y 74.137,Z 230.000,A 0.000,B 0.000,C 180.000,E1 0.000} C_DIS
LIN {X -151.941,Y 66.403,Z 230.000,A 0.000,B 0.000,C 180.000,E1 0.000} C_DIS
LIN {X -155.159,Y 58.491,Z 230.000,A 0.000,B 0.000,C 180.000,E1 0.000} C_DIS
LIN {X -155.711,Y 56.905,Z 230.000,A 0.000,B 0.000,C 180.000,E1 0.000} C_DIS
LIN {X -157.964,Y 50.427,Z 230.000,A 0.000,B 0.000,C 180.000,E1 0.000} C_DIS
LIN {X -160.351,Y 42.229,Z 230.000,A 0.000,B 0.000,C 180.000,E1 0.000} C_DIS
LIN {X -162.312,Y 33.919,Z 230.000,A 0.000,B 0.000,C 180.000,E1 0.000} C_DIS
LIN {X -163.843,Y 25.518,Z 230.000,A 0.000,B 0.000,C 180.000,E1 0.000} C_DIS
LIN {X -164.939,Y 17.048,Z 230.000,A 0.000,B 0.000,C 180.000,E1 0.000} C_DIS
LIN {X -165.598,Y 8.536,Z 230.000,A 0.000,B 0.000,C 180.000,E1 0.000} C_DIS
LIN {X -165.818,Y 0.000,Z 230.000,A 0.000,B 0.000,C 180.000,E1 0.000} C_DIS
LIN {X -165.598,Y -8.536,Z 230.000,A 0.000,B 0.000,C 180.000,E1 0.000} C_DIS
LIN {X -164.939,Y -17.048,Z 230.000,A 0.000,B 0.000,C 180.000,E1 0.000} C_DIS
LIN {X -163.843,Y -25.518,Z 230.000,A 0.000,B 0.000,C 180.000,E1 0.000} C_DIS
LIN {X -162.312,Y -33.919,Z 230.000,A 0.000,B 0.000,C 180.000,E1 0.000} C_DIS
LIN {X -160.351,Y -42.229,Z 230.000,A 0.000,B 0.000,C 180.000,E1 0.000} C_DIS
LIN {X -157.964,Y -50.427,Z 230.000,A 0.000,B 0.000,C 180.000,E1 0.000} C_DIS
LIN {X -155.158,Y -58.493,Z 230.000,A 0.000,B 0.000,C 180.000,E1 0.000} C_DIS
LIN {X -151.941,Y -66.403,Z 230.000,A 0.000,B 0.000,C 180.000,E1 0.000} C_DIS
LIN {X -148.322,Y -74.137,Z 230.000,A 0.000,B 0.000,C 180.000,E1 0.000} C_DIS
LIN {X -144.309,Y -81.674,Z 230.000,A 0.000,B 0.000,C 180.000,E1 0.000} C_DIS
LIN {X -139.913,Y -88.994,Z 230.000,A 0.000,B 0.000,C 180.000,E1 0.000} C_DIS
LIN {X -135.146,Y -96.079,Z 230.000,A 0.000,B 0.000,C 180.000,E1 0.000} C_DIS
LIN {X -130.022,Y -102.908,Z 230.000,A 0.000,B 0.000,C 180.000,E1 0.000} C_DIS
LIN {X -124.551,Y -109.465,Z 230.000,A 0.000,B 0.000,C 180.000,E1 0.000} C_DIS
LIN {X -118.751,Y -115.732,Z 230.000,A 0.000,B 0.000,C 180.000,E1 0.000} C_DIS
LIN {X -112.636,Y -121.692,Z 230.000,A 0.000,B 0.000,C 180.000,E1 0.000} C_DIS
LIN {X -106.222,Y -127.329,Z 230.000,A 0.000,B 0.000,C 180.000,E1 0.000} C_DIS
LIN {X -99.526,Y -132.628,Z 230.000,A 0.000,B 0.000,C 180.000,E1 0.000} C_DIS
LIN {X -92.567,Y -137.576,Z 230.000,A 0.000,B 0.000,C 180.000,E1 0.000} C_DIS
LIN {X -85.363,Y -142.157,Z 230.000,A 0.000,B 0.000,C 180.000,E1 0.000} C_DIS
LIN {X -77.930,Y -146.364,Z 230.000,A 0.000,B 0.000,C 180.000,E1 0.000} C_DIS
LIN {X -70.292,Y -150.183,Z 230.000,A 0.000,B 0.000,C 180.000,E1 0.000} C_DIS
LIN {X -62.470,Y -153.601,Z 230.000,A 0.000,B 0.000,C 180.000,E1 0.000} C_DIS
LIN {X -54.479,Y -156.612,Z 230.000,A 0.000,B 0.000,C 180.000,E1 0.000} C_DIS
LIN {X -46.343,Y -159.210,Z 230.000,A 0.000,B 0.000,C 180.000,E1 0.000} C_DIS
LIN {X -38.086,Y -161.385,Z 230.000,A 0.000,B 0.000,C 180.000,E1 0.000} C_DIS
LIN {X -29.728,Y -163.132,Z 230.000,A 0.000,B 0.000,C 180.000,E1 0.000} C_DIS
LIN {X -21.292,Y -164.446,Z 230.000,A 0.000,B 0.000,C 180.000,E1 0.000} C_DIS
LIN {X -12.798,Y -165.324,Z 230.000,A 0.000,B 0.000,C 180.000,E1 0.000} C_DIS
LIN {X -4.269,Y -165.763,Z 230.000,A 0.000,B 0.000,C 180.000,E1 0.000} C_DIS
LIN {X 4.269,Y -165.763,Z 230.000,A 0.000,B 0.000,C 180.000,E1 0.000} C_DIS
LIN {X 12.798,Y -165.324,Z 230.000,A 0.000,B 0.000,C 180.000,E1 0.000} C_DIS
LIN {X 21.292,Y -164.446,Z 230.000,A 0.000,B 0.000,C 180.000,E1 0.000} C_DIS
LIN {X 29.728,Y -163.132,Z 230.000,A 0.000,B 0.000,C 180.000,E1 0.000} C_DIS
LIN {X 38.087,Y -161.385,Z 230.000,A 0.000,B 0.000,C 180.000,E1 0.000} C_DIS
LIN {X 46.343,Y -159.210,Z 230.000,A 0.000,B 0.000,C 180.000,E1 0.000} C_DIS
LIN {X 54.479,Y -156.612,Z 230.000,A 0.000,B 0.000,C 180.000,E1 0.000} C_DIS
LIN {X 62.470,Y -153.601,Z 230.000,A 0.000,B 0.000,C 180.000,E1 0.000} C_DIS
LIN {X 70.292,Y -150.183,Z 230.000,A 0.000,B 0.000,C 180.000,E1 0.000} C_DIS
LIN {X 77.930,Y -146.364,Z 230.000,A 0.000,B 0.000,C 180.000,E1 0.000} C_DIS
LIN {X 85.363,Y -142.157,Z 230.000,A 0.000,B 0.000,C 180.000,E1 0.000} C_DIS
LIN {X 92.567,Y -137.576,Z 230.000,A 0.000,B 0.000,C 180.000,E1 0.000} C_DIS
LIN {X 99.526,Y -132.628,Z 230.000,A 0.000,B 0.000,C 180.000,E1 0.000} C_DIS
LIN {X 106.222,Y -127.329,Z 230.000,A 0.000,B 0.000,C 180.000,E1 0.000} C_DIS
LIN {X 112.636,Y -121.692,Z 230.000,A 0.000,B 0.000,C 180.000,E1 0.000} C_DIS
LIN {X 118.751,Y -115.732,Z 230.000,A 0.000,B 0.000,C 180.000,E1 0.000} C_DIS
LIN {X 124.551,Y -109.465,Z 230.000,A 0.000,B 0.000,C 180.000,E1 0.000} C_DIS
LIN {X 130.022,Y -102.908,Z 230.000,A 0.000,B 0.000,C 180.000,E1 0.000} C_DIS
LIN {X 135.146,Y -96.079,Z 230.000,A 0.000,B 0.000,C 180.000,E1 0.000} C_DIS
LIN {X 139.913,Y -88.994,Z 230.000,A 0.000,B 0.000,C 180.000,E1 0.000} C_DIS
LIN {X 144.309,Y -81.673,Z 230.000,A 0.000,B 0.000,C 180.000,E1 0.000} C_DIS
LIN {X 148.322,Y -74.137,Z 230.000,A 0.000,B 0.000,C 180.000,E1 0.000} C_DIS
LIN {X 151.941,Y -66.403,Z 230.000,A 0.000,B 0.000,C 180.000,E1 0.000} C_DIS
LIN {X 155.159,Y -58.491,Z 230.000,A 0.000,B 0.000,C 180.000,E1 0.000} C_DIS
LIN {X 157.964,Y -50.427,Z 230.000,A 0.000,B 0.000,C 180.000,E1 0.000} C_DIS
LIN {X 160.351,Y -42.229,Z 230.000,A 0.000,B 0.000,C 180.000,E1 0.000} C_DIS
LIN {X 162.312,Y -33.919,Z 230.000,A 0.000,B 0.000,C 180.000,E1 0.000} C_DIS
LIN {X 163.843,Y -25.518,Z 230.000,A 0.000,B 0.000,C 180.000,E1 0.000} C_DIS
LIN {X 164.939,Y -17.048,Z 230.000,A 0.000,B 0.000,C 180.000,E1 0.000} C_DIS
LIN {X 165.598,Y -8.536,Z 230.000,A 0.000,B 0.000,C 180.000,E1 0.000} C_DIS
LIN {X 165.818,Y 0.000,Z 230.000,A 0.000,B 0.000,C 180.000,E1 0.000} C_DIS
LIN {X 165.598,Y 8.536,Z 230.000,A 0.000,B 0.000,C 180.000,E1 0.000} C_DIS
;rapid-leaky
$VEL.CP=0.3
LIN {X 146.523,Y -20.971,Z 230.000,A 0.000,B 0.000,C 180.000,E1 0.000} C_DIS
;bead-sparse_infill
$VEL.CP=0.41
LIN {X -20.970,Y 146.522,Z 230.000,A 0.000,B 0.000,C 180.000,E1 0.000} C_DIS
LIN {X -26.543,Y 145.654,Z 230.000,A 0.000,B 0.000,C 180.000,E1 0.000} C_DIS
LIN {X -34.005,Y 144.094,Z 230.000,A 0.000,B 0.000,C 180.000,E1 0.000} C_DIS
LIN {X -41.377,Y 142.153,Z 230.000,A 0.000,B 0.000,C 180.000,E1 0.000} C_DIS
LIN {X -48.643,Y 139.833,Z 230.000,A 0.000,B 0.000,C 180.000,E1 0.000} C_DIS
LIN {X -55.778,Y 137.144,Z 230.000,A 0.000,B 0.000,C 180.000,E1 0.000} C_DIS
LIN {X -62.760,Y 134.092,Z 230.000,A 0.000,B 0.000,C 180.000,E1 0.000} C_DIS
LIN {X -69.579,Y 130.683,Z 230.000,A 0.000,B 0.000,C 180.000,E1 0.000} C_DIS
LIN {X -76.218,Y 126.926,Z 230.000,A 0.000,B 0.000,C 180.000,E1 0.000} C_DIS
LIN {X -82.650,Y 122.835,Z 230.000,A 0.000,B 0.000,C 180.000,E1 0.000} C_DIS
LIN {X -88.863,Y 118.418,Z 230.000,A 0.000,B 0.000,C 180.000,E1 0.000} C_DIS
LIN {X -94.842,Y 113.686,Z 230.000,A 0.000,B 0.000,C 180.000,E1 0.000} C_DIS
LIN {X -100.568,Y 108.654,Z 230.000,A 0.000,B 0.000,C 180.000,E1 0.000} C_DIS
LIN {X -106.027,Y 103.333,Z 230.000,A 0.000,B 0.000,C 180.000,E1 0.000} C_DIS
LIN {X -111.207,Y 97.737,Z 230.000,A 0.000,B 0.000,C 180.000,E1 0.000} C_DIS
LIN {X -116.092,Y 91.882,Z 230.000,A 0.000,B 0.000,C 180.000,E1 0.000} C_DIS
LIN {X -119.185,Y 87.759,Z 230.000,A 0.000,B 0.000,C 180.000,E1 0.000} C_DIS
LIN {X 87.770,Y -119.195,Z 230.000,A 0.000,B 0.000,C 180.000,E1 0.000} C_DIS
LIN {X 82.650,Y -122.835,Z 230.000,A 0.000,B 0.000,C 180.000,E1 0.000} C_DIS
LIN {X 76.218,Y -126.926,Z 230.000,A 0.000,B 0.000,C 180.000,E1 0.000} C_DIS
LIN {X 69.579,Y -130.683,Z 230.000,A 0.000,B 0.000,C 180.000,E1 0.000} C_DIS
LIN {X 62.760,Y -134.092,Z 230.000,A 0.000,B 0.000,C 180.000,E1 0.000} C_DIS
LIN {X 55.778,Y -137.144,Z 230.000,A 0.000,B 0.000,C 180.000,E1 0.000} C_DIS
LIN {X 48.643,Y -139.833,Z 230.000,A 0.000,B 0.000,C 180.000,E1 0.000} C_DIS
LIN {X 41.377,Y -142.153,Z 230.000,A 0.000,B 0.000,C 180.000,E1 0.000} C_DIS
LIN {X 34.005,Y -144.094,Z 230.000,A 0.000,B 0.000,C 180.000,E1 0.000} C_DIS
LIN {X 26.543,Y -145.654,Z 230.000,A 0.000,B 0.000,C 180.000,E1 0.000} C_DIS
LIN {X 19.011,Y -146.827,Z 230.000,A 0.000,B 0.000,C 180.000,E1 0.000} C_DIS
LIN {X 11.427,Y -147.611,Z 230.000,A 0.000,B 0.000,C 180.000,E1 0.000} C_DIS
LIN {X 3.812,Y -148.003,Z 230.000,A 0.000,B 0.000,C 180.000,E1 0.000} C_DIS
LIN {X -3.812,Y -148.003,Z 230.000,A 0.000,B 0.000,C 180.000,E1 0.000} C_DIS
LIN {X -11.427,Y -147.611,Z 230.000,A 0.000,B 0.000,C 180.000,E1 0.000} C_DIS
LIN {X -19.011,Y -146.827,Z 230.000,A 0.000,B 0.000,C 180.000,E1 0.000} C_DIS
LIN {X -26.543,Y -145.654,Z 230.000,A 0.000,B 0.000,C 180.000,E1 0.000} C_DIS
LIN {X -34.005,Y -144.094,Z 230.000,A 0.000,B 0.000,C 180.000,E1 0.000} C_DIS
LIN {X -41.377,Y -142.153,Z 230.000,A 0.000,B 0.000,C 180.000,E1 0.000} C_DIS
LIN {X -48.537,Y -139.866,Z 230.000,A 0.000,B 0.000,C 180.000,E1 0.000} C_DIS
LIN {X -139.791,Y -48.613,Z 230.000,A 0.000,B 0.000,C 180.000,E1 0.000} C_DIS
;rapid-leaky
$VEL.CP=0.3
LIN {X 165.149,Y 34.511,Z 240.000,A 0.000,B 0.000,C 180.000,E1 0.000} C_DIS
;bead-perimeter_outer
$VEL.CP=0.37
LIN {X 163.153,Y 42.967,Z 240.000,A 0.000,B 0.000,C 180.000,E1 0.000} C_DIS
LIN {X 160.725,Y 51.309,Z 240.000,A 0.000,B 0.000,C 180.000,E1 0.000} C_DIS
LIN {X 157.871,Y 59.515,Z 240.000,A 0.000,B 0.000,C 180.000,E1 0.000} C_DIS
LIN {X 154.597,Y 67.564,Z 240.000,A 0.000,B 0.000,C 180.000,E1 0.000} C_DIS
LIN {X 153.556,Y 69.790,Z 240.000,A 0.000,B 0.000,C 180.000,E1 0.000} C_DIS
LIN {X 150.915,Y 75.432,Z 240.000,A 0.000,B 0.000,C 180.000,E1 0.000} C_DIS
LIN {X 146.832,Y 83.101,Z 240.000,A 0.000,B 0.000,C 180.000,E1 0.000} C_DIS
LIN {X 142.359,Y 90.549,Z 240.000,A 0.000,B 0.000,C 180.000,E1 0.000} C_DIS
LIN {X 137.509,Y 97.757,Z 240.000,A 0.000,B 0.000,C 180.000,E1 0.000} C_DIS
LIN {X 132.293,Y 104.707,Z 240.000,A 0.000,B 0.000,C 180.000,E1 0.000} C_DIS
LIN {X 126.729,Y 111.379,Z 240.000,A 0.000,B 0.000,C 180.000,E1 0.000} C_DIS
LIN {X 120.826,Y 117.755,Z 240.000,A 0.000,B 0.000,C 180.000,E1 0.000} C_DIS
LIN {X 114.605,Y 123.819,Z 240.000,A 0.000,B 0.000,C 180.000,E1 0.000} C_DIS
LIN {X 108.079,Y 129.553,Z 240.000,A 0.000,B 0.000,C 180.000,E1 0.000} C_DIS
LIN {X 101.265,Y 134.946,Z 240.000,A 0.000,B 0.000,C 180.000,E1 0.000} C_DIS
LIN {X 94.184,Y 139.981,Z 240.000,A 0.000,B 0.000,C 180.000,E1 0.000} C_DIS
LIN {X 86.854,Y 144.643,Z 240.000,A 0.000,B 0.000,C 180.000,E1 0.000} C_DIS
LIN {X 79.293,Y 148.923,Z 240.000,A 0.000,B 0.000,C 180.000,E1 0.000} C_DIS
LIN {X 71.521,Y 152.807,Z 240.000,A 0.000,B 0.000,C 180.000,E1 0.000} C_DIS
LIN {X 63.559,Y 156.287,Z 240.000,A 0.000,B 0.000,C 180.000,E1 0.000} C_DIS
LIN {X 55.432,Y 159.350,Z 240.000,A 0.000,B 0.000,C 180.000,E1 0.000} C_DIS
LIN {X 47.154,Y 161.993,Z 240.000,A 0.000,B 0.000,C 180.000,E1 0.000} C_DIS
LIN {X 38.752,Y 164.205,Z 240.000,A 0.000,B 0.000,C 180.000,E1 0.000} C_DIS
LIN {X 30.247,Y 165.983,Z 240.000,A 0.000,B 0.000,C 180.000,E1 0.000} C_DIS
LIN {X 21.663,Y 167.320,Z 240.000,A 0.000,B 0.000,C 180.000,E1 0.000} C_DIS
LIN {X 13.021,Y 168.213,Z 240.000,A 0.000,B 0.000,C 180.000,E1 0.000} C_DIS
LIN {X 4.344,Y 168.661,Z 240.000,A 0.000,B 0.000,C 180.000,E1 0.000} C_DIS
LIN {X -4.344,Y 168.661,Z 240.000,A 0.000,B 0.000,C 180.000,E1 0.000} C_DIS
LIN {X -13.021,Y 168.213,Z 240.000,A 0.000,B 0.000,C 180.000,E1 0.000} C_DIS
LIN {X -21.663,Y 167.320,Z 240.000,A 0.000,B 0.000,C 180.000,E1 0.000} C_DIS
LIN {X -30.247,Y 165.983,Z 240.000,A 0.000,B 0.000,C 180.000,E1 0.000} C_DIS
LIN {X -38.752,Y 164.205,Z 240.000,A 0.000,B 0.000,C 180.000,E1 0.000} C_DIS
LIN {X -47.154,Y 161.993,Z 240.000,A 0.000,B 0.000,C 180.000,E1 0.000} C_DIS
LIN {X -55.431,Y 159.351,Z 240.000,A 0.000,B 0.000,C 180.000,E1 0.000} C_DIS
LIN {X -63.560,Y 156.286,Z 240.000,A 0.000,B 0.000,C 180.000,E1 0.000} C_DIS
LIN {X -71.521,Y 152.807,Z 240.000,A 0.000,B 0.000,C 180.000,E1 0.000} C_DIS
LIN {X -79.293,Y 148.923,Z 240.000,A 0.000,B 0.000,C 180.000,E1 0.000} C_DIS
LIN {X -86.854,Y 144.643,Z 240.000,A 0.000,B 0.000,C 180.000,E1 0.000} C_DIS
LIN {X -94.184,Y 139.981,Z 240.000,A 0.000,B 0.000,C 180.000,E1 0.000} C_DIS
LIN {X -101.265,Y 134.946,Z 240.000,A 0.000,B 0.000,C 180.000,E1 0.000} C_DIS
LIN {X -108.079,Y 129.553,Z 240.000,A 0.000,B 0.000,C 180.000,E1 0.000} C_DIS
LIN {X -114.605,Y 123.819,Z 240.000,A 0.000,B 0.000,C 180.000,E1 0.000} C_DIS
LIN {X -120.826,Y 117.755,Z 240.000,A 0.000,B 0.000,C 180.000,E1 0.000} C_DIS
LIN {X -126.729,Y 111.379,Z 240.000,A 0.000,B 0.000,C 180.000,E1 0.000} C_DIS
LIN {X -132.293,Y 104.707,Z 240.000,A 0.000,B 0.000,C 180.000,E1 0.000} C_DIS
LIN {X -137.509,Y 97.757,Z 240.000,A 0.000,B 0.000,C 180.000,E1 0.000} C_DIS
LIN {X -142.359,Y 90.549,Z 240.000,A 0.000,B 0.000,C 180.000,E1 0.000} C_DIS
LIN {X -146.832,Y 83.101,Z 240.000,A 0.000,B 0.000,C 180.000,E1 0.000} C_DIS
LIN {X -150.915,Y 75.433,Z 240.000,A 0.000,B 0.000,C 180.000,E1 0.000} C_DIS
LIN {X -154.598,Y 67.564,Z 240.000,A 0.000,B 0.000,C 180.000,E1 0.000} C_DIS
LIN {X -157.871,Y 59.515,Z 240.000,A 0.000,B 0.000,C 180.000,E1 0.000} C_DIS
LIN {X -160.725,Y 51.309,Z 240.000,A 0.000,B 0.000,C 180.000,E1 0.000} C_DIS
LIN {X -163.153,Y 42.967,Z 240.000,A 0.000,B 0.000,C 180.000,E1 0.000} C_DIS
LIN {X -165.149,Y 34.511,Z 240.000,A 0.000,B 0.000,C 180.000,E1 0.000} C_DIS
LIN {X -166.707,Y 25.964,Z 240.000,A 0.000,B 0.000,C 180.000,E1 0.000} C_DIS
LIN {X -167.822,Y 17.347,Z 240.000,A 0.000,B 0.000,C 180.000,E1 0.000} C_DIS
LIN {X -168.493,Y 8.685,Z 240.000,A 0.000,B 0.000,C 180.000,E1 0.000} C_DIS
LIN {X -168.716,Y 0.000,Z 240.000,A 0.000,B 0.000,C 180.000,E1 0.000} C_DIS
LIN {X -168.493,Y -8.685,Z 240.000,A 0.000,B 0.000,C 180.000,E1 0.000} C_DIS
LIN {X -167.822,Y -17.347,Z 240.000,A 0.000,B 0.000,C 180.000,E1 0.000} C_DIS
LIN {X -166.707,Y -25.964,Z 240.000,A 0.000,B 0.000,C 180.000,E1 0.000} C_DIS
LIN {X -165.149,Y -34.511,Z 240.000,A 0.000,B 0.000,C 180.000,E1 0.000} C_DIS
LIN {X -163.153,Y -42.967,Z 240.000,A 0.000,B 0.000,C 180.000,E1 0.000} C_DIS
LIN {X -160.725,Y -51.309,Z 240.000,A 0.000,B 0.000,C 180.000,E1 0.000} C_DIS
LIN {X -157.871,Y -59.515,Z 240.000,A 0.000,B 0.000,C 180.000,E1 0.000} C_DIS
LIN {X -154.597,Y -67.564,Z 240.000,A 0.000,B 0.000,C 180.000,E1 0.000} C_DIS
LIN {X -150.915,Y -75.432,Z 240.000,A 0.000,B 0.000,C 180.000,E1 0.000} C_DIS
LIN {X -146.832,Y -83.101,Z 240.000,A 0.000,B 0.000,C 180.000,E1 0.000} C_DIS
LIN {X -142.359,Y -90.549,Z 240.000,A 0.000,B 0.000,C 180.000,E1 0.000} C_DIS
LIN {X -137.509,Y -97.757,Z 240.000,A 0.000,B 0.000,C 180.000,E1 0.000} C_DIS
LIN {X -132.293,Y -104.707,Z 240.000,A 0.000,B 0.000,C 180.000,E1 0.000} C_DIS
LIN {X -126.729,Y -111.379,Z 240.000,A 0.000,B 0.000,C 180.000,E1 0.000} C_DIS
LIN {X -120.826,Y -117.755,Z 240.000,A 0.000,B 0.000,C 180.000,E1 0.000} C_DIS
LIN {X -114.605,Y -123.819,Z 240.000,A 0.000,B 0.000,C 180.000,E1 0.000} C_DIS
LIN {X -108.079,Y -129.553,Z 240.000,A 0.000,B 0.000,C 180.000,E1 0.000} C_DIS
LIN {X -101.265,Y -134.946,Z 240.000,A 0.000,B 0.000,C 180.000,E1 0.000} C_DIS
LIN {X -94.184,Y -139.981,Z 240.000,A 0.000,B 0.000,C 180.000,E1 0.000} C_DIS
LIN {X -86.854,Y -144.643,Z 240.000,A 0.000,B 0.000,C 180.000,E1 0.000} C_DIS
LIN {X -79.293,Y -148.923,Z 240.000,A 0.000,B 0.000,C 180.000,E1 0.000} C_DIS
LIN {X -71.521,Y -152.807,Z 240.000,A 0.000,B 0.000,C 180.000,E1 0.000} C_DIS
LIN {X -63.559,Y -156.287,Z 240.000,A 0.000,B 0.000,C 180.000,E1 0.000} C_DIS
LIN {X -55.432,Y -159.350,Z 240.000,A 0.000,B 0.000,C 180.000,E1 0.000} C_DIS
LIN {X -47.154,Y -161.993,Z 240.000,A 0.000,B 0.000,C 180.000,E1 0.000} C_DIS
LIN {X -38.752,Y -164.205,Z 240.000,A 0.000,B 0.000,C 180.000,E1 0.000} C_DIS
LIN {X -30.247,Y -165.983,Z 240.000,A 0.000,B 0.000,C 180.000,E1 0.000} C_DIS
LIN {X -21.663,Y -167.320,Z 240.000,A 0.000,B 0.000,C 180.000,E1 0.000} C_DIS
LIN {X -13.021,Y -168.213,Z 240.000,A 0.000,B 0.000,C 180.000,E1 0.000} C_DIS
LIN {X -4.344,Y -168.661,Z 240.000,A 0.000,B 0.000,C 180.000,E1 0.000} C_DIS
LIN {X 4.344,Y -168.661,Z 240.000,A 0.000,B 0.000,C 180.000,E1 0.000} C_DIS
LIN {X 13.021,Y -168.213,Z 240.000,A 0.000,B 0.000,C 180.000,E1 0.000} C_DIS
LIN {X 21.663,Y -167.320,Z 240.000,A 0.000,B 0.000,C 180.000,E1 0.000} C_DIS
LIN {X 30.247,Y -165.983,Z 240.000,A 0.000,B 0.000,C 180.000,E1 0.000} C_DIS
LIN {X 38.752,Y -164.205,Z 240.000,A 0.000,B 0.000,C 180.000,E1 0.000} C_DIS
LIN {X 47.154,Y -161.993,Z 240.000,A 0.000,B 0.000,C 180.000,E1 0.000} C_DIS
LIN {X 55.431,Y -159.351,Z 240.000,A 0.000,B 0.000,C 180.000,E1 0.000} C_DIS
LIN {X 63.560,Y -156.286,Z 240.000,A 0.000,B 0.000,C 180.000,E1 0.000} C_DIS
LIN {X 71.521,Y -152.807,Z 240.000,A 0.000,B 0.000,C 180.000,E1 0.000} C_DIS
LIN {X 79.293,Y -148.923,Z 240.000,A 0.000,B 0.000,C 180.000,E1 0.000} C_DIS
LIN {X 86.854,Y -144.643,Z 240.000,A 0.000,B 0.000,C 180.000,E1 0.000} C_DIS
LIN {X 94.184,Y -139.981,Z 240.000,A 0.000,B 0.000,C 180.000,E1 0.000} C_DIS
LIN {X 101.265,Y -134.946,Z 240.000,A 0.000,B 0.000,C 180.000,E1 0.000} C_DIS
LIN {X 108.079,Y -129.553,Z 240.000,A 0.000,B 0.000,C 180.000,E1 0.000} C_DIS
LIN {X 114.605,Y -123.819,Z 240.000,A 0.000,B 0.000,C 180.000,E1 0.000} C_DIS
LIN {X 120.826,Y -117.755,Z 240.000,A 0.000,B 0.000,C 180.000,E1 0.000} C_DIS
LIN {X 126.729,Y -111.379,Z 240.000,A 0.000,B 0.000,C 180.000,E1 0.000} C_DIS
LIN {X 132.293,Y -104.707,Z 240.000,A 0.000,B 0.000,C 180.000,E1 0.000} C_DIS
LIN {X 137.509,Y -97.757,Z 240.000,A 0.000,B 0.000,C 180.000,E1 0.000} C_DIS
LIN {X 142.359,Y -90.549,Z 240.000,A 0.000,B 0.000,C 180.000,E1 0.000} C_DIS
LIN {X 146.832,Y -83.101,Z 240.000,A 0.000,B 0.000,C 180.000,E1 0.000} C_DIS
LIN {X 150.915,Y -75.433,Z 240.000,A 0.000,B 0.000,C 180.000,E1 0.000} C_DIS
LIN {X 154.598,Y -67.564,Z 240.000,A 0.000,B 0.000,C 180.000,E1 0.000} C_DIS
LIN {X 157.871,Y -59.515,Z 240.000,A 0.000,B 0.000,C 180.000,E1 0.000} C_DIS
LIN {X 160.725,Y -51.309,Z 240.000,A 0.000,B 0.000,C 180.000,E1 0.000} C_DIS
LIN {X 163.153,Y -42.967,Z 240.000,A 0.000,B 0.000,C 180.000,E1 0.000} C_DIS
LIN {X 165.149,Y -34.511,Z 240.000,A 0.000,B 0.000,C 180.000,E1 0.000} C_DIS
LIN {X 166.707,Y -25.964,Z 240.000,A 0.000,B 0.000,C 180.000,E1 0.000} C_DIS
LIN {X 167.822,Y -17.347,Z 240.000,A 0.000,B 0.000,C 180.000,E1 0.000} C_DIS
LIN {X 168.493,Y -8.685,Z 240.000,A 0.000,B 0.000,C 180.000,E1 0.000} C_DIS
LIN {X 168.716,Y 0.000,Z 240.000,A 0.000,B 0.000,C 180.000,E1 0.000} C_DIS
LIN {X 168.493,Y 8.685,Z 240.000,A 0.000,B 0.000,C 180.000,E1 0.000} C_DIS
LIN {X 167.822,Y 17.347,Z 240.000,A 0.000,B 0.000,C 180.000,E1 0.000} C_DIS
LIN {X 166.707,Y 25.964,Z 240.000,A 0.000,B 0.000,C 180.000,E1 0.000} C_DIS
LIN {X 165.149,Y 34.511,Z 240.000,A 0.000,B 0.000,C 180.000,E1 0.000} C_DIS
;rapid-leaky
$VEL.CP=0.3
LIN {X 149.933,Y 31.331,Z 240.000,A 0.000,B 0.000,C 180.000,E1 0.000} C_DIS
;bead-perimeter_inner
$VEL.CP=0.37
LIN {X 148.121,Y 39.008,Z 240.000,A 0.000,B 0.000,C 180.000,E1 0.000} C_DIS
LIN {X 145.916,Y 46.582,Z 240.000,A 0.000,B 0.000,C 180.000,E1 0.000} C_DIS
LIN {X 143.325,Y 54.031,Z 240.000,A 0.000,B 0.000,C 180.000,E1 0.000} C_DIS
LIN {X 140.352,Y 61.340,Z 240.000,A 0.000,B 0.000,C 180.000,E1 0.000} C_DIS
LIN {X 139.481,Y 63.203,Z 240.000,A 0.000,B 0.000,C 180.000,E1 0.000} C_DIS
LIN {X 137.010,Y 68.482,Z 240.000,A 0.000,B 0.000,C 180.000,E1 0.000} C_DIS
LIN {X 133.303,Y 75.443,Z 240.000,A 0.000,B 0.000,C 180.000,E1 0.000} C_DIS
LIN {X 129.242,Y 82.206,Z 240.000,A 0.000,B 0.000,C 180.000,E1 0.000} C_DIS
LIN {X 124.840,Y 88.750,Z 240.000,A 0.000,B 0.000,C 180.000,E1 0.000} C_DIS
LIN {X 120.104,Y 95.060,Z 240.000,A 0.000,B 0.000,C 180.000,E1 0.000} C_DIS
LIN {X 115.052,Y 101.117,Z 240.000,A 0.000,B 0.000,C 180.000,E1 0.000} C_DIS
LIN {X 109.694,Y 106.905,Z 240.000,A 0.000,B 0.000,C 180.000,E1 0.000} C_DIS
LIN {X 104.046,Y 112.410,Z 240.000,A 0.000,B 0.000,C 180.000,E1 0.000} C_DIS
LIN {X 98.121,Y 117.616,Z 240.000,A 0.000,B 0.000,C 180.000,E1 0.000} C_DIS
LIN {X 91.934,Y 122.513,Z 240.000,A 0.000,B 0.000,C 180.000,E1 0.000} C_DIS
LIN {X 85.506,Y 127.083,Z 240.000,A 0.000,B 0.000,C 180.000,E1 0.000} C_DIS
LIN {X 78.850,Y 131.316,Z 240.000,A 0.000,B 0.000,C 180.000,E1 0.000} C_DIS
LIN {X 71.987,Y 135.202,Z 240.000,A 0.000,B 0.000,C 180.000,E1 0.000} C_DIS
LIN {X 64.932,Y 138.728,Z 240.000,A 0.000,B 0.000,C 180.000,E1 0.000} C_DIS
LIN {X 57.702,Y 141.887,Z 240.000,A 0.000,B 0.000,C 180.000,E1 0.000} C_DIS
LIN {X 50.325,Y 144.668,Z 240.000,A 0.000,B 0.000,C 180.000,E1 0.000} C_DIS
LIN {X 42.809,Y 147.067,Z 240.000,A 0.000,B 0.000,C 180.000,E1 0.000} C_DIS
LIN {X 35.181,Y 149.076,Z 240.000,A 0.000,B 0.000,C 180.000,E1 0.000} C_DIS
LIN {X 27.459,Y 150.690,Z 240.000,A 0.000,B 0.000,C 180.000,E1 0.000} C_DIS
LIN {X 19.667,Y 151.904,Z 240.000,A 0.000,B 0.000,C 180.000,E1 0.000} C_DIS
LIN {X 11.821,Y 152.715,Z 240.000,A 0.000,B 0.000,C 180.000,E1 0.000} C_DIS
LIN {X 3.943,Y 153.121,Z 240.000,A 0.000,B 0.000,C 180.000,E1 0.000} C_DIS
LIN {X -3.943,Y 153.121,Z 240.000,A 0.000,B 0.000,C 180.000,E1 0.000} C_DIS
LIN {X -11.821,Y 152.715,Z 240.000,A 0.000,B 0.000,C 180.000,E1 0.000} C_DIS
LIN {X -19.667,Y 151.904,Z 240.000,A 0.000,B 0.000,C 180.000,E1 0.000} C_DIS
LIN {X -27.459,Y 150.690,Z 240.000,A 0.000,B 0.000,C 180.000,E1 0.000} C_DIS
LIN {X -35.181,Y 149.076,Z 240.000,A 0.000,B 0.000,C 180.000,E1 0.000} C_DIS
LIN {X -42.809,Y 147.067,Z 240.000,A 0.000,B 0.000,C 180.000,E1 0.000} C_DIS
LIN {X -50.324,Y 144.668,Z 240.000,A 0.000,B 0.000,C 180.000,E1 0.000} C_DIS
LIN {X -57.704,Y 141.886,Z 240.000,A 0.000,B 0.000,C 180.000,E1 0.000} C_DIS
LIN {X -64.932,Y 138.728,Z 240.000,A 0.000,B 0.000,C 180.000,E1 0.000} C_DIS
LIN {X -71.987,Y 135.202,Z 240.000,A 0.000,B 0.000,C 180.000,E1 0.000} C_DIS
LIN {X -78.850,Y 131.316,Z 240.000,A 0.000,B 0.000,C 180.000,E1 0.000} C_DIS
LIN {X -85.506,Y 127.083,Z 240.000,A 0.000,B 0.000,C 180.000,E1 0.000} C_DIS
LIN {X -91.934,Y 122.513,Z 240.000,A 0.000,B 0.000,C 180.000,E1 0.000} C_DIS
LIN {X -98.121,Y 117.616,Z 240.000,A 0.000,B 0.000,C 180.000,E1 0.000} C_DIS
LIN {X -104.046,Y 112.410,Z 240.000,A 0.000,B 0.000,C 180.000,E1 0.000} C_DIS
LIN {X -109.694,Y 106.905,Z 240.000,A 0.000,B 0.000,C 180.000,E1 0.000} C_DIS
LIN {X -115.052,Y 101.117,Z 240.000,A 0.000,B 0.000,C 180.000,E1 0.000} C_DIS
LIN {X -120.104,Y 95.060,Z 240.000,A 0.000,B 0.000,C 180.000,E1 0.000} C_DIS
LIN {X -124.840,Y 88.750,Z 240.000,A 0.000,B 0.000,C 180.000,E1 0.000} C_DIS
LIN {X -129.242,Y 82.206,Z 240.000,A 0.000,B 0.000,C 180.000,E1 0.000} C_DIS
LIN {X -133.303,Y 75.443,Z 240.000,A 0.000,B 0.000,C 180.000,E1 0.000} C_DIS
LIN {X -137.010,Y 68.483,Z 240.000,A 0.000,B 0.000,C 180.000,E1 0.000} C_DIS
LIN {X -140.353,Y 61.339,Z 240.000,A 0.000,B 0.000,C 180.000,E1 0.000} C_DIS
LIN {X -143.325,Y 54.031,Z 240.000,A 0.000,B 0.000,C 180.000,E1 0.000} C_DIS
LIN {X -145.916,Y 46.582,Z 240.000,A 0.000,B 0.000,C 180.000,E1 0.000} C_DIS
LIN {X -148.121,Y 39.008,Z 240.000,A 0.000,B 0.000,C 180.000,E1 0.000} C_DIS
LIN {X -149.933,Y 31.331,Z 240.000,A 0.000,B 0.000,C 180.000,E1 0.000} C_DIS
LIN {X -151.347,Y 23.572,Z 240.000,A 0.000,B 0.000,C 180.000,E1 0.000} C_DIS
LIN {X -152.359,Y 15.748,Z 240.000,A 0.000,B 0.000,C 180.000,E1 0.000} C_DIS
LIN {X -152.968,Y 7.885,Z 240.000,A 0.000,B 0.000,C 180.000,E1 0.000} C_DIS
LIN {X -153.171,Y 0.000,Z 240.000,A 0.000,B 0.000,C 180.000,E1 0.000} C_DIS
LIN {X -152.968,Y -7.885,Z 240.000,A 0.000,B 0.000,C 180.000,E1 0.000} C_DIS
LIN {X -152.359,Y -15.748,Z 240.000,A 0.000,B 0.000,C 180.000,E1 0.000} C_DIS
LIN {X -151.347,Y -23.572,Z 240.000,A 0.000,B 0.000,C 180.000,E1 0.000} C_DIS
LIN {X -149.933,Y -31.331,Z 240.000,A 0.000,B 0.000,C 180.000,E1 0.000} C_DIS
LIN {X -148.121,Y -39.008,Z 240.000,A 0.000,B 0.000,C 180.000,E1 0.000} C_DIS
LIN {X -145.916,Y -46.582,Z 240.000,A 0.000,B 0.000,C 180.000,E1 0.000} C_DIS
LIN {X -143.325,Y -54.031,Z 240.000,A 0.000,B 0.000,C 180.000,E1 0.000} C_DIS
LIN {X -140.352,Y -61.340,Z 240.000,A 0.000,B 0.000,C 180.000,E1 0.000} C_DIS
LIN {X -137.010,Y -68.482,Z 240.000,A 0.000,B 0.000,C 180.000,E1 0.000} C_DIS
LIN {X -133.303,Y -75.443,Z 240.000,A 0.000,B 0.000,C 180.000,E1 0.000} C_DIS
LIN {X -129.242,Y -82.206,Z 240.000,A 0.000,B 0.000,C 180.000,E1 0.000} C_DIS
LIN {X -124.840,Y -88.750,Z 240.000,A 0.000,B 0.000,C 180.000,E1 0.000} C_DIS
LIN {X -120.104,Y -95.060,Z 240.000,A 0.000,B 0.000,C 180.000,E1 0.000} C_DIS
LIN {X -115.052,Y -101.117,Z 240.000,A 0.000,B 0.000,C 180.000,E1 0.000} C_DIS
LIN {X -109.694,Y -106.905,Z 240.000,A 0.000,B 0.000,C 180.000,E1 0.000} C_DIS
LIN {X -104.046,Y -112.410,Z 240.000,A 0.000,B 0.000,C 180.000,E1 0.000} C_DIS
LIN {X -98.121,Y -117.616,Z 240.000,A 0.000,B 0.000,C 180.000,E1 0.000} C_DIS
LIN {X -91.934,Y -122.513,Z 240.000,A 0.000,B 0.000,C 180.000,E1 0.000} C_DIS
LIN {X -85.506,Y -127.083,Z 240.000,A 0.000,B 0.000,C 180.000,E1 0.000} C_DIS
LIN {X -78.850,Y -131.316,Z 240.000,A 0.000,B 0.000,C 180.000,E1 0.000} C_DIS
LIN {X -71.987,Y -135.202,Z 240.000,A 0.000,B 0.000,C 180.000,E1 0.000} C_DIS
LIN {X -64.932,Y -138.728,Z 240.000,A 0.000,B 0.000,C 180.000,E1 0.000} C_DIS
LIN {X -57.702,Y -141.887,Z 240.000,A 0.000,B 0.000,C 180.000,E1 0.000} C_DIS
LIN {X -50.325,Y -144.668,Z 240.000,A 0.000,B 0.000,C 180.000,E1 0.000} C_DIS
LIN {X -42.809,Y -147.067,Z 240.000,A 0.000,B 0.000,C 180.000,E1 0.000} C_DIS
LIN {X -35.181,Y -149.076,Z 240.000,A 0.000,B 0.000,C 180.000,E1 0.000} C_DIS
LIN {X -27.459,Y -150.690,Z 240.000,A 0.000,B 0.000,C 180.000,E1 0.000} C_DIS
LIN {X -19.667,Y -151.904,Z 240.000,A 0.000,B 0.000,C 180.000,E1 0.000} C_DIS
LIN {X -11.821,Y -152.715,Z 240.000,A 0.000,B 0.000,C 180.000,E1 0.000} C_DIS
LIN {X -3.943,Y -153.121,Z 240.000,A 0.000,B 0.000,C 180.000,E1 0.000} C_DIS
LIN {X 3.943,Y -153.121,Z 240.000,A 0.000,B 0.000,C 180.000,E1 0.000} C_DIS
LIN {X 11.821,Y -152.715,Z 240.000,A 0.000,B 0.000,C 180.000,E1 0.000} C_DIS
LIN {X 19.667,Y -151.904,Z 240.000,A 0.000,B 0.000,C 180.000,E1 0.000} C_DIS
LIN {X 27.459,Y -150.690,Z 240.000,A 0.000,B 0.000,C 180.000,E1 0.000} C_DIS
LIN {X 35.181,Y -149.076,Z 240.000,A 0.000,B 0.000,C 180.000,E1 0.000} C_DIS
LIN {X 42.809,Y -147.067,Z 240.000,A 0.000,B 0.000,C 180.000,E1 0.000} C_DIS
LIN {X 50.324,Y -144.668,Z 240.000,A 0.000,B 0.000,C 180.000,E1 0.000} C_DIS
LIN {X 57.704,Y -141.886,Z 240.000,A 0.000,B 0.000,C 180.000,E1 0.000} C_DIS
LIN {X 64.932,Y -138.728,Z 240.000,A 0.000,B 0.000,C 180.000,E1 0.000} C_DIS
LIN {X 71.987,Y -135.202,Z 240.000,A 0.000,B 0.000,C 180.000,E1 0.000} C_DIS
LIN {X 78.850,Y -131.316,Z 240.000,A 0.000,B 0.000,C 180.000,E1 0.000} C_DIS
LIN {X 85.506,Y -127.083,Z 240.000,A 0.000,B 0.000,C 180.000,E1 0.000} C_DIS
LIN {X 91.934,Y -122.513,Z 240.000,A 0.000,B 0.000,C 180.000,E1 0.000} C_DIS
LIN {X 98.121,Y -117.616,Z 240.000,A 0.000,B 0.000,C 180.000,E1 0.000} C_DIS
LIN {X 104.046,Y -112.410,Z 240.000,A 0.000,B 0.000,C 180.000,E1 0.000} C_DIS
LIN {X 109.694,Y -106.905,Z 240.000,A 0.000,B 0.000,C 180.000,E1 0.000} C_DIS
LIN {X 115.052,Y -101.117,Z 240.000,A 0.000,B 0.000,C 180.000,E1 0.000} C_DIS
LIN {X 120.104,Y -95.060,Z 240.000,A 0.000,B 0.000,C 180.000,E1 0.000} C_DIS
LIN {X 124.840,Y -88.750,Z 240.000,A 0.000,B 0.000,C 180.000,E1 0.000} C_DIS
LIN {X 129.242,Y -82.206,Z 240.000,A 0.000,B 0.000,C 180.000,E1 0.000} C_DIS
LIN {X 133.303,Y -75.443,Z 240.000,A 0.000,B 0.000,C 180.000,E1 0.000} C_DIS
LIN {X 137.010,Y -68.483,Z 240.000,A 0.000,B 0.000,C 180.000,E1 0.000} C_DIS
LIN {X 140.353,Y -61.339,Z 240.000,A 0.000,B 0.000,C 180.000,E1 0.000} C_DIS
LIN {X 143.325,Y -54.031,Z 240.000,A 0.000,B 0.000,C 180.000,E1 0.000} C_DIS
LIN {X 145.916,Y -46.582,Z 240.000,A 0.000,B 0.000,C 180.000,E1 0.000} C_DIS
LIN {X 148.121,Y -39.008,Z 240.000,A 0.000,B 0.000,C 180.000,E1 0.000} C_DIS
LIN {X 149.933,Y -31.331,Z 240.000,A 0.000,B 0.000,C 180.000,E1 0.000} C_DIS
LIN {X 151.347,Y -23.572,Z 240.000,A 0.000,B 0.000,C 180.000,E1 0.000} C_DIS
LIN {X 152.359,Y -15.748,Z 240.000,A 0.000,B 0.000,C 180.000,E1 0.000} C_DIS
LIN {X 152.968,Y -7.885,Z 240.000,A 0.000,B 0.000,C 180.000,E1 0.000} C_DIS
LIN {X 153.171,Y 0.000,Z 240.000,A 0.000,B 0.000,C 180.000,E1 0.000} C_DIS
LIN {X 152.968,Y 7.885,Z 240.000,A 0.000,B 0.000,C 180.000,E1 0.000} C_DIS
LIN {X 152.359,Y 15.748,Z 240.000,A 0.000,B 0.000,C 180.000,E1 0.000} C_DIS
LIN {X 151.347,Y 23.572,Z 240.000,A 0.000,B 0.000,C 180.000,E1 0.000} C_DIS
LIN {X 149.933,Y 31.331,Z 240.000,A 0.000,B 0.000,C 180.000,E1 0.000} C_DIS
;rapid-leaky
$VEL.CP=0.3
LIN {X -9.499,Y -135.051,Z 240.000,A 0.000,B 0.000,C 180.000,E1 0.000} C_DIS
;bead-sparse_infill
$VEL.CP=0.37
LIN {X 135.032,Y 9.480,Z 240.000,A 0.000,B 0.000,C 180.000,E1 0.000} C_DIS
LIN {X 134.688,Y 13.921,Z 240.000,A 0.000,B 0.000,C 180.000,E1 0.000} C_DIS
LIN {X 133.792,Y 20.838,Z 240.000,A 0.000,B 0.000,C 180.000,E1 0.000} C_DIS
LIN {X 132.542,Y 27.697,Z 240.000,A 0.000,B 0.000,C 180.000,E1 0.000} C_DIS
LIN {X 130.941,Y 34.484,Z 240.000,A 0.000,B 0.000,C 180.000,E1 0.000} C_DIS
LIN {X 128.992,Y 41.180,Z 240.000,A 0.000,B 0.000,C 180.000,E1 0.000} C_DIS
LIN {X 126.701,Y 47.764,Z 240.000,A 0.000,B 0.000,C 180.000,E1 0.000} C_DIS
LIN {X 124.073,Y 54.227,Z 240.000,A 0.000,B 0.000,C 180.000,E1 0.000} C_DIS
LIN {X 123.396,Y 55.673,Z 240.000,A 0.000,B 0.000,C 180.000,E1 0.000} C_DIS
LIN {X 121.119,Y 60.539,Z 240.000,A 0.000,B 0.000,C 180.000,E1 0.000} C_DIS
LIN {X 117.842,Y 66.692,Z 240.000,A 0.000,B 0.000,C 180.000,E1 0.000} C_DIS
LIN {X 114.252,Y 72.671,Z 240.000,A 0.000,B 0.000,C 180.000,E1 0.000} C_DIS
LIN {X 110.360,Y 78.456,Z 240.000,A 0.000,B 0.000,C 180.000,E1 0.000} C_DIS
LIN {X 106.173,Y 84.035,Z 240.000,A 0.000,B 0.000,C 180.000,E1 0.000} C_DIS
LIN {X 101.707,Y 89.389,Z 240.000,A 0.000,B 0.000,C 180.000,E1 0.000} C_DIS
LIN {X 96.971,Y 94.506,Z 240.000,A 0.000,B 0.000,C 180.000,E1 0.000} C_DIS
LIN {X 91.978,Y 99.372,Z 240.000,A 0.000,B 0.000,C 180.000,E1 0.000} C_DIS
LIN {X 86.741,Y 103.973,Z 240.000,A 0.000,B 0.000,C 180.000,E1 0.000} C_DIS
LIN {X 81.270,Y 108.303,Z 240.000,A 0.000,B 0.000,C 180.000,E1 0.000} C_DIS
LIN {X 78.703,Y 110.129,Z 240.000,A 0.000,B 0.000,C 180.000,E1 0.000} C_DIS
LIN {X -110.155,Y -78.729,Z 240.000,A 0.000,B 0.000,C 180.000,E1 0.000} C_DIS
LIN {X -110.360,Y -78.456,Z 240.000,A 0.000,B 0.000,C 180.000,E1 0.000} C_DIS
LIN {X -114.252,Y -72.671,Z 240.000,A 0.000,B 0.000,C 180.000,E1 0.000} C_DIS
LIN {X -117.842,Y -66.692,Z 240.000,A 0.000,B 0.000,C 180.000,E1 0.000} C_DIS
LIN {X -121.119,Y -60.539,Z 240.000,A 0.000,B 0.000,C 180.000,E1 0.000} C_DIS
LIN {X -124.073,Y -54.226,Z 240.000,A 0.000,B 0.000,C 180.000,E1 0.000} C_DIS
LIN {X -126.701,Y -47.764,Z 240.000,A 0.000,B 0.000,C 180.000,E1 0.000} C_DIS
LIN {X -128.992,Y -41.180,Z 240.000,A 0.000,B 0.000,C 180.000,E1 0.000} C_DIS
LIN {X -130.941,Y -34.484,Z 240.000,A 0.000,B 0.000,C 180.000,E1 0.000} C_DIS
LIN {X -132.542,Y -27.697,Z 240.000,A 0.000,B 0.000,C 180.000,E1 0.000} C_DIS
LIN {X -133.792,Y -20.838,Z 240.000,A 0.000,B 0.000,C 180.000,E1 0.000} C_DIS
LIN {X -134.688,Y -13.921,Z 240.000,A 0.000,B 0.000,C 180.000,E1 0.000} C_DIS
LIN {X -135.226,Y -6.971,Z 240.000,A 0.000,B 0.000,C 180.000,E1 0.000} C_DIS
LIN {X -135.405,Y 0.000,Z 240.000,A 0.000,B 0.000,C 180.000,E1 0.000} C_DIS
LIN {X -135.226,Y 6.971,Z 240.000,A 0.000,B 0.000,C 180.000,E1 0.000} C_DIS
LIN {X -134.688,Y 13.921,Z 240.000,A 0.000,B 0.000,C 180.000,E1 0.000} C_DIS
LIN {X -133.792,Y 20.838,Z 240.000,A 0.000,B 0.000,C 180.000,E1 0.000} C_DIS
LIN {X -132.542,Y 27.697,Z 240.000,A 0.000,B 0.000,C 180.000,E1 0.000} C_DIS
LIN {X -130.941,Y 34.484,Z 240.000,A 0.000,B 0.000,C 180.000,E1 0.000} C_DIS
LIN {X -128.992,Y 41.180,Z 240.000,A 0.000,B 0.000,C 180.000,E1 0.000} C_DIS
LIN {X -126.701,Y 47.764,Z 240.000,A 0.000,B 0.000,C 180.000,E1 0.000} C_DIS
LIN {X -124.074,Y 54.224,Z 240.000,A 0.000,B 0.000,C 180.000,E1 0.000} C_DIS
LIN {X -121.118,Y 60.540,Z 240.000,A 0.000,B 0.000,C 180.000,E1 0.000} C_DIS
LIN {X -117.842,Y 66.692,Z 240.000,A 0.000,B 0.000,C 180.000,E1 0.000} C_DIS
LIN {X -114.252,Y 72.671,Z 240.000,A 0.000,B 0.000,C 180.000,E1 0.000} C_DIS
LIN {X -111.207,Y 77.196,Z 240.000,A 0.000,B 0.000,C 180.000,E1 0.000} C_DIS
LIN {X -77.221,Y 111.182,Z 240.000,A 0.000,B 0.000,C 180.000,E1 0.000} C_DIS
;rapid-leaky
$VEL.CP=0.3
LIN {X -138.230,Y 69.091,Z 250.000,A 0.000,B 0.000,C 180.000,E1 0.000} C_DIS
;bead-perimeter_outer
$VEL.CP=0.32
LIN {X -141.604,Y 61.884,Z 250.000,A 0.000,B 0.000,C 180.000,E1 0.000} C_DIS
LIN {X -144.602,Y 54.513,Z 250.000,A 0.000,B 0.000,C 180.000,E1 0.000} C_DIS
LIN {X -147.216,Y 46.996,Z 250.000,A 0.000,B 0.000,C 180.000,E1 0.000} C_DIS
LIN {X -149.440,Y 39.356,Z 250.000,A 0.000,B 0.000,C 180.000,E1 0.000} C_DIS
LIN {X -151.268,Y 31.611,Z 250.000,A 0.000,B 0.000,C 180.000,E1 0.000} C_DIS
LIN {X -152.695,Y 23.781,Z 250.000,A 0.000,B 0.000,C 180.000,E1 0.000} C_DIS
LIN {X -153.716,Y 15.890,Z 250.000,A 0.000,B 0.000,C 180.000,E1 0.000} C_DIS
LIN {X -154.331,Y 7.955,Z 250.000,A 0.000,B 0.000,C 180.000,E1 0.000} C_DIS
LIN {X -154.535,Y 0.000,Z 250.000,A 0.000,B 0.000,C 180.000,E1 0.000} C_DIS
LIN {X -154.331,Y -7.955,Z 250.000,A 0.000,B 0.000,C 180.000,E1 0.000} C_DIS
LIN {X -153.716,Y -15.890,Z 250.000,A 0.000,B 0.000,C 180.000,E1 0.000} C_DIS
LIN {X -152.695,Y -23.781,Z 250.000,A 0.000,B 0.000,C 180.000,E1 0.000} C_DIS
LIN {X -151.268,Y -31.611,Z 250.000,A 0.000,B 0.000,C 180.000,E1 0.000} C_DIS
LIN {X -149.440,Y -39.356,Z 250.000,A 0.000,B 0.000,C 180.000,E1 0.000} C_DIS
LIN {X -147.216,Y -46.996,Z 250.000,A 0.000,B 0.000,C 180.000,E1 0.000} C_DIS
LIN {X -144.602,Y -54.513,Z 250.000,A 0.000,B 0.000,C 180.000,E1 0.000} C_DIS
LIN {X -141.604,Y -61.884,Z 250.000,A 0.000,B 0.000,C 180.000,E1 0.000} C_DIS
LIN {X -140.158,Y -64.973,Z 250.000,A 0.000,B 0.000,C 180.000,E1 0.000} C_DIS
LIN {X -138.230,Y -69.091,Z 250.000,A 0.000,B 0.000,C 180.000,E1 0.000} C_DIS
LIN {X -134.490,Y -76.116,Z 250.000,A 0.000,B 0.000,C 180.000,E1 0.000} C_DIS
LIN {X -130.393,Y -82.939,Z 250.000,A 0.000,B 0.000,C 180.000,E1 0.000} C_DIS
LIN {X -125.951,Y -89.541,Z 250.000,A 0.000,B 0.000,C 180.000,E1 0.000} C_DIS
LIN {X -121.175,Y -95.906,Z 250.000,A 0.000,B 0.000,C 180.000,E1 0.000} C_DIS
LIN {X -116.077,Y -102.017,Z 250.000,A 0.000,B 0.000,C 180.000,E1 0.000} C_DIS
LIN {X -110.671,Y -107.857,Z 250.000,A 0.000,B 0.000,C 180.000,E1 0.000} C_DIS
LIN {X -104.972,Y -113.412,Z 250.000,A 0.000,B 0.000,C 180.000,E1 0.000} C_DIS
LIN {X -98.994,Y -118.665,Z 250.000,A 0.000,B 0.000,C 180.000,E1 0.000} C_DIS
LIN {X -92.754,Y -123.604,Z 250.000,A 0.000,B 0.000,C 180.000,E1 0.000} C_DIS
LIN {X -86.268,Y -128.215,Z 250.000,A 0.000,B 0.000,C 180.000,E1 0.000} C_DIS
LIN {X -79.554,Y -132.486,Z 250.000,A 0.000,B 0.000,C 180.000,E1 0.000} C_DIS
LIN {X -72.628,Y -136.405,Z 250.000,A 0.000,B 0.000,C 180.000,E1 0.000} C_DIS
LIN {X -65.510,Y -139.963,Z 250.000,A 0.000,B 0.000,C 180.000,E1 0.000} C_DIS
LIN {X -58.218,Y -143.150,Z 250.000,A 0.000,B 0.000,C 180.000,E1 0.000} C_DIS
LIN {X -50.773,Y -145.956,Z 250.000,A 0.000,B 0.000,C 180.000,E1 0.000} C_DIS
LIN {X -43.189,Y -148.377,Z 250.000,A 0.000,B 0.000,C 180.000,E1 0.000} C_DIS
LIN {X -35.494,Y -150.404,Z 250.000,A 0.000,B 0.000,C 180.000,E1 0.000} C_DIS
LIN {X -27.706,Y -152.032,Z 250.000,A 0.000,B 0.000,C 180.000,E1 0.000} C_DIS
LIN {X -19.843,Y -153.256,Z 250.000,A 0.000,B 0.000,C 180.000,E1 0.000} C_DIS
LIN {X -11.926,Y -154.074,Z 250.000,A 0.000,B 0.000,C 180.000,E1 0.000} C_DIS
LIN {X -3.978,Y -154.485,Z 250.000,A 0.000,B 0.000,C 180.000,E1 0.000} C_DIS
LIN {X 3.978,Y -154.485,Z 250.000,A 0.000,B 0.000,C 180.000,E1 0.000} C_DIS
LIN {X 11.926,Y -154.074,Z 250.000,A 0.000,B 0.000,C 180.000,E1 0.000} C_DIS
LIN {X 19.843,Y -153.256,Z 250.000,A 0.000,B 0.000,C 180.000,E1 0.000} C_DIS
LIN {X 27.706,Y -152.032,Z 250.000,A 0.000,B 0.000,C 180.000,E1 0.000} C_DIS
LIN {X 35.494,Y -150.404,Z 250.000,A 0.000,B 0.000,C 180.000,E1 0.000} C_DIS
LIN {X 43.189,Y -148.377,Z 250.000,A 0.000,B 0.000,C 180.000,E1 0.000} C_DIS
LIN {X 50.773,Y -145.956,Z 250.000,A 0.000,B 0.000,C 180.000,E1 0.000} C_DIS
LIN {X 58.218,Y -143.150,Z 250.000,A 0.000,B 0.000,C 180.000,E1 0.000} C_DIS
LIN {X 65.510,Y -139.963,Z 250.000,A 0.000,B 0.000,C 180.000,E1 0.000} C_DIS
LIN {X 72.628,Y -136.405,Z 250.000,A 0.000,B 0.000,C 180.000,E1 0.000} C_DIS
LIN {X 79.554,Y -132.486,Z 250.000,A 0.000,B 0.000,C 180.000,E1 0.000} C_DIS
LIN {X 86.268,Y -128.215,Z 250.000,A 0.000,B 0.000,C 180.000,E1 0.000} C_DIS
LIN {X 92.754,Y -123.604,Z 250.000,A 0.000,B 0.000,C 180.000,E1 0.000} C_DIS
LIN {X 98.994,Y -118.665,Z 250.000,A 0.000,B 0.000,C 180.000,E1 0.000} C_DIS
LIN {X 104.972,Y -113.412,Z 250.000,A 0.000,B 0.000,C 180.000,E1 0.000} C_DIS
LIN {X 110.671,Y -107.857,Z 250.000,A 0.000,B 0.000,C 180.000,E1 0.000} C_DIS
LIN {X 116.077,Y -102.017,Z 250.000,A 0.000,B 0.000,C 180.000,E1 0.000} C_DIS
LIN {X 121.175,Y -95.906,Z 250.000,A 0.000,B 0.000,C 180.000,E1 0.000} C_DIS
LIN {X 125.951,Y -89.541,Z 250.000,A 0.000,B 0.000,C 180.000,E1 0.000} C_DIS
LIN {X 130.393,Y -82.939,Z 250.000,A 0.000,B 0.000,C 180.000,E1 0.000} C_DIS
LIN {X 134.490,Y -76.116,Z 250.000,A 0.000,B 0.000,C 180.000,E1 0.000} C_DIS
LIN {X 138.230,Y -69.091,Z 250.000,A 0.000,B 0.000,C 180.000,E1 0.000} C_DIS
LIN {X 141.604,Y -61.884,Z 250.000,A 0.000,B 0.000,C 180.000,E1 0.000} C_DIS
LIN {X 144.602,Y -54.513,Z 250.000,A 0.000,B 0.000,C 180.000,E1 0.000} C_DIS
LIN {X 147.216,Y -46.996,Z 250.000,A 0.000,B 0.000,C 180.000,E1 0.000} C_DIS
LIN {X 149.440,Y -39.356,Z 250.000,A 0.000,B 0.000,C 180.000,E1 0.000} C_DIS
LIN {X 151.268,Y -31.611,Z 250.000,A 0.000,B 0.000,C 180.000,E1 0.000} C_DIS
LIN {X 152.695,Y -23.781,Z 250.000,A 0.000,B 0.000,C 180.000,E1 0.000} C_DIS
LIN {X 153.716,Y -15.890,Z 250.000,A 0.000,B 0.000,C 180.000,E1 0.000} C_DIS
LIN {X 154.331,Y -7.955,Z 250.000,A 0.000,B 0.000,C 180.000,E1 0.000} C_DIS
LIN {X 154.535,Y 0.000,Z 250.000,A 0.000,B 0.000,C 180.000,E1 0.000} C_DIS
LIN {X 154.331,Y 7.955,Z 250.000,A 0.000,B 0.000,C 180.000,E1 0.000} C_DIS
LIN {X 153.716,Y 15.890,Z 250.000,A 0.000,B 0.000,C 180.000,E1 0.000} C_DIS
LIN {X 152.695,Y 23.781,Z 250.000,A 0.000,B 0.000,C 180.000,E1 0.000} C_DIS
LIN {X 151.268,Y 31.611,Z 250.000,A 0.000,B 0.000,C 180.000,E1 0.000} C_DIS
LIN {X 149.440,Y 39.356,Z 250.000,A 0.000,B 0.000,C 180.000,E1 0.000} C_DIS
LIN {X 147.216,Y 46.996,Z 250.000,A 0.000,B 0.000,C 180.000,E1 0.000} C_DIS
LIN {X 144.602,Y 54.513,Z 250.000,A 0.000,B 0.000,C 180.000,E1 0.000} C_DIS
LIN {X 141.604,Y 61.884,Z 250.000,A 0.000,B 0.000,C 180.000,E1 0.000} C_DIS
LIN {X 138.230,Y 69.091,Z 250.000,A 0.000,B 0.000,C 180.000,E1 0.000} C_DIS
LIN {X 134.490,Y 76.116,Z 250.000,A 0.000,B 0.000,C 180.000,E1 0.000} C_DIS
LIN {X 130.393,Y 82.939,Z 250.000,A 0.000,B 0.000,C 180.000,E1 0.000} C_DIS
LIN {X 125.951,Y 89.541,Z 250.000,A 0.000,B 0.000,C 180.000,E1 0.000} C_DIS
LIN {X 121.175,Y 95.906,Z 250.000,A 0.000,B 0.000,C 180.000,E1 0.000} C_DIS
LIN {X 116.077,Y 102.017,Z 250.000,A 0.000,B 0.000,C 180.000,E1 0.000} C_DIS
LIN {X 110.671,Y 107.857,Z 250.000,A 0.000,B 0.000,C 180.000,E1 0.000} C_DIS
LIN {X 104.972,Y 113.412,Z 250.000,A 0.000,B 0.000,C 180.000,E1 0.000} C_DIS
LIN {X 98.994,Y 118.665,Z 250.000,A 0.000,B 0.000,C 180.000,E1 0.000} C_DIS
LIN {X 92.754,Y 123.604,Z 250.000,A 0.000,B 0.000,C 180.000,E1 0.000} C_DIS
LIN {X 86.268,Y 128.215,Z 250.000,A 0.000,B 0.000,C 180.000,E1 0.000} C_DIS
LIN {X 79.554,Y 132.486,Z 250.000,A 0.000,B 0.000,C 180.000,E1 0.000} C_DIS
LIN {X 72.628,Y 136.405,Z 250.000,A 0.000,B 0.000,C 180.000,E1 0.000} C_DIS
LIN {X 65.510,Y 139.963,Z 250.000,A 0.000,B 0.000,C 180.000,E1 0.000} C_DIS
LIN {X 58.218,Y 143.150,Z 250.000,A 0.000,B 0.000,C 180.000,E1 0.000} C_DIS
LIN {X 50.773,Y 145.956,Z 250.000,A 0.000,B 0.000,C 180.000,E1 0.000} C_DIS
LIN {X 43.189,Y 148.377,Z 250.000,A 0.000,B 0.000,C 180.000,E1 0.000} C_DIS
LIN {X 35.494,Y 150.404,Z 250.000,A 0.000,B 0.000,C 180.000,E1 0.000} C_DIS
LIN {X 27.706,Y 152.032,Z 250.000,A 0.000,B 0.000,C 180.000,E1 0.000} C_DIS
LIN {X 19.843,Y 153.256,Z 250.000,A 0.000,B 0.000,C 180.000,E1 0.000} C_DIS
LIN {X 11.926,Y 154.074,Z 250.000,A 0.000,B 0.000,C 180.000,E1 0.000} C_DIS
LIN {X 3.978,Y 154.485,Z 250.000,A 0.000,B 0.000,C 180.000,E1 0.000} C_DIS
LIN {X -3.978,Y 154.485,Z 250.000,A 0.000,B 0.000,C 180.000,E1 0.000} C_DIS
LIN {X -11.926,Y 154.074,Z 250.000,A 0.000,B 0.000,C 180.000,E1 0.000} C_DIS
LIN {X -19.843,Y 153.256,Z 250.000,A 0.000,B 0.000,C 180.000,E1 0.000} C_DIS
LIN {X -27.706,Y 152.032,Z 250.000,A 0.000,B 0.000,C 180.000,E1 0.000} C_DIS
LIN {X -35.494,Y 150.404,Z 250.000,A 0.000,B 0.000,C 180.000,E1 0.000} C_DIS
LIN {X -43.189,Y 148.377,Z 250.000,A 0.000,B 0.000,C 180.000,E1 0.000} C_DIS
LIN {X -50.773,Y 145.956,Z 250.000,A 0.000,B 0.000,C 180.000,E1 0.000} C_DIS
LIN {X -58.218,Y 143.150,Z 250.000,A 0.000,B 0.000,C 180.000,E1 0.000} C_DIS
LIN {X -65.510,Y 139.963,Z 250.000,A 0.000,B 0.000,C 180.000,E1 0.000} C_DIS
LIN {X -72.628,Y 136.405,Z 250.000,A 0.000,B 0.000,C 180.000,E1 0.000} C_DIS
LIN {X -79.554,Y 132.486,Z 250.000,A 0.000,B 0.000,C 180.000,E1 0.000} C_DIS
LIN {X -86.268,Y 128.215,Z 250.000,A 0.000,B 0.000,C 180.000,E1 0.000} C_DIS
LIN {X -92.754,Y 123.604,Z 250.000,A 0.000,B 0.000,C 180.000,E1 0.000} C_DIS
LIN {X -98.994,Y 118.665,Z 250.000,A 0.000,B 0.000,C 180.000,E1 0.000} C_DIS
LIN {X -104.972,Y 113.412,Z 250.000,A 0.000,B 0.000,C 180.000,E1 0.000} C_DIS
LIN {X -110.671,Y 107.857,Z 250.000,A 0.000,B 0.000,C 180.000,E1 0.000} C_DIS
LIN {X -116.077,Y 102.017,Z 250.000,A 0.000,B 0.000,C 180.000,E1 0.000} C_DIS
LIN {X -121.175,Y 95.906,Z 250.000,A 0.000,B 0.000,C 180.000,E1 0.000} C_DIS
LIN {X -125.951,Y 89.541,Z 250.000,A 0.000,B 0.000,C 180.000,E1 0.000} C_DIS
LIN {X -130.393,Y 82.939,Z 250.000,A 0.000,B 0.000,C 180.000,E1 0.000} C_DIS
LIN {X -134.490,Y 76.116,Z 250.000,A 0.000,B 0.000,C 180.000,E1 0.000} C_DIS
LIN {X -138.230,Y 69.091,Z 250.000,A 0.000,B 0.000,C 180.000,E1 0.000} C_DIS
;rapid-leaky
$VEL.CP=0.3
LIN {X -124.325,Y 62.141,Z 250.000,A 0.000,B 0.000,C 180.000,E1 0.000} C_DIS
;bead-perimeter_inner
$VEL.CP=0.32
LIN {X -127.360,Y 55.658,Z 250.000,A 0.000,B 0.000,C 180.000,E1 0.000} C_DIS
LIN {X -130.056,Y 49.029,Z 250.000,A 0.000,B 0.000,C 180.000,E1 0.000} C_DIS
LIN {X -132.407,Y 42.269,Z 250.000,A 0.000,B 0.000,C 180.000,E1 0.000} C_DIS
LIN {X -134.408,Y 35.397,Z 250.000,A 0.000,B 0.000,C 180.000,E1 0.000} C_DIS
LIN {X -136.051,Y 28.432,Z 250.000,A 0.000,B 0.000,C 180.000,E1 0.000} C_DIS
LIN {X -137.335,Y 21.390,Z 250.000,A 0.000,B 0.000,C 180.000,E1 0.000} C_DIS
LIN {X -138.254,Y 14.291,Z 250.000,A 0.000,B 0.000,C 180.000,E1 0.000} C_DIS
LIN {X -138.806,Y 7.155,Z 250.000,A 0.000,B 0.000,C 180.000,E1 0.000} C_DIS
LIN {X -138.990,Y 0.000,Z 250.000,A 0.000,B 0.000,C 180.000,E1 0.000} C_DIS
LIN {X -138.806,Y -7.155,Z 250.000,A 0.000,B 0.000,C 180.000,E1 0.000} C_DIS
LIN {X -138.254,Y -14.291,Z 250.000,A 0.000,B 0.000,C 180.000,E1 0.000} C_DIS
LIN {X -137.335,Y -21.390,Z 250.000,A 0.000,B 0.000,C 180.000,E1 0.000} C_DIS
LIN {X -136.051,Y -28.432,Z 250.000,A 0.000,B 0.000,C 180.000,E1 0.000} C_DIS
LIN {X -134.408,Y -35.397,Z 250.000,A 0.000,B 0.000,C 180.000,E1 0.000} C_DIS
LIN {X -132.407,Y -42.269,Z 250.000,A 0.000,B 0.000,C 180.000,E1 0.000} C_DIS
LIN {X -130.056,Y -49.029,Z 250.000,A 0.000,B 0.000,C 180.000,E1 0.000} C_DIS
LIN {X -127.360,Y -55.659,Z 250.000,A 0.000,B 0.000,C 180.000,E1 0.000} C_DIS
LIN {X -126.084,Y -58.384,Z 250.000,A 0.000,B 0.000,C 180.000,E1 0.000} C_DIS
LIN {X -124.326,Y -62.140,Z 250.000,A 0.000,B 0.000,C 180.000,E1 0.000} C_DIS
LIN {X -120.961,Y -68.459,Z 250.000,A 0.000,B 0.000,C 180.000,E1 0.000} C_DIS
LIN {X -117.276,Y -74.597,Z 250.000,A 0.000,B 0.000,C 180.000,E1 0.000} C_DIS
LIN {X -113.281,Y -80.534,Z 250.000,A 0.000,B 0.000,C 180.000,E1 0.000} C_DIS
LIN {X -108.985,Y -86.258,Z 250.000,A 0.000,B 0.000,C 180.000,E1 0.000} C_DIS
LIN {X -104.400,Y -91.755,Z 250.000,A 0.000,B 0.000,C 180.000,E1 0.000} C_DIS
LIN {X -99.538,Y -97.008,Z 250.000,A 0.000,B 0.000,C 180.000,E1 0.000} C_DIS
LIN {X -94.413,Y -102.003,Z 250.000,A 0.000,B 0.000,C 180.000,E1 0.000} C_DIS
LIN {X -89.036,Y -106.728,Z 250.000,A 0.000,B 0.000,C 180.000,E1 0.000} C_DIS
LIN {X -83.424,Y -111.170,Z 250.000,A 0.000,B 0.000,C 180.000,E1 0.000} C_DIS
LIN {X -77.591,Y -115.317,Z 250.000,A 0.000,B 0.000,C 180.000,E1 0.000} C_DIS
LIN {X -71.551,Y -119.159,Z 250.000,A 0.000,B 0.000,C 180.000,E1 0.000} C_DIS
LIN {X -65.322,Y -122.684,Z 250.000,A 0.000,B 0.000,C 180.000,E1 0.000} C_DIS
LIN {X -58.920,Y -125.884,Z 250.000,A 0.000,B 0.000,C 180.000,E1 0.000} C_DIS
LIN {X -52.361,Y -128.751,Z 250.000,A 0.000,B 0.000,C 180.000,E1 0.000} C_DIS
LIN {X -45.667,Y -131.274,Z 250.000,A 0.000,B 0.000,C 180.000,E1 0.000} C_DIS
LIN {X -38.844,Y -133.451,Z 250.000,A 0.000,B 0.000,C 180.000,E1 0.000} C_DIS
LIN {X -31.922,Y -135.275,Z 250.000,A 0.000,B 0.000,C 180.000,E1 0.000} C_DIS
LIN {X -24.919,Y -136.739,Z 250.000,A 0.000,B 0.000,C 180.000,E1 0.000} C_DIS
LIN {X -17.847,Y -137.840,Z 250.000,A 0.000,B 0.000,C 180.000,E1 0.000} C_DIS
LIN {X -10.725,Y -138.576,Z 250.000,A 0.000,B 0.000,C 180.000,E1 0.000} C_DIS
LIN {X -3.577,Y -138.945,Z 250.000,A 0.000,B 0.000,C 180.000,E1 0.000} C_DIS
LIN {X 3.577,Y -138.945,Z 250.000,A 0.000,B 0.000,C 180.000,E1 0.000} C_DIS
LIN {X 10.725,Y -138.576,Z 250.000,A 0.000,B 0.000,C 180.000,E1 0.000} C_DIS
LIN {X 17.847,Y -137.840,Z 250.000,A 0.000,B 0.000,C 180.000,E1 0.000} C_DIS
LIN {X 24.920,Y -136.739,Z 250.000,A 0.000,B 0.000,C 180.000,E1 0.000} C_DIS
LIN {X 31.922,Y -135.275,Z 250.000,A 0.000,B 0.000,C 180.000,E1 0.000} C_DIS
LIN {X 38.844,Y -133.451,Z 250.000,A 0.000,B 0.000,C 180.000,E1 0.000} C_DIS
LIN {X 45.666,Y -131.274,Z 250.000,A 0.000,B 0.000,C 180.000,E1 0.000} C_DIS
LIN {X 52.362,Y -128.750,Z 250.000,A 0.000,B 0.000,C 180.000,E1 0.000} C_DIS
LIN {X 58.920,Y -125.884,Z 250.000,A 0.000,B 0.000,C 180.000,E1 0.000} C_DIS
LIN {X 65.322,Y -122.684,Z 250.000,A 0.000,B 0.000,C 180.000,E1 0.000} C_DIS
LIN {X 71.551,Y -119.159,Z 250.000,A 0.000,B 0.000,C 180.000,E1 0.000} C_DIS
LIN {X 77.591,Y -115.317,Z 250.000,A 0.000,B 0.000,C 180.000,E1 0.000} C_DIS
LIN {X 83.424,Y -111.170,Z 250.000,A 0.000,B 0.000,C 180.000,E1 0.000} C_DIS
LIN {X 89.036,Y -106.728,Z 250.000,A 0.000,B 0.000,C 180.000,E1 0.000} C_DIS
LIN {X 94.413,Y -102.003,Z 250.000,A 0.000,B 0.000,C 180.000,E1 0.000} C_DIS
LIN {X 99.538,Y -97.008,Z 250.000,A 0.000,B 0.000,C 180.000,E1 0.000} C_DIS
LIN {X 104.400,Y -91.755,Z 250.000,A 0.000,B 0.000,C 180.000,E1 0.000} C_DIS
LIN {X 108.985,Y -86.258,Z 250.000,A 0.000,B 0.000,C 180.000,E1 0.000} C_DIS
LIN {X 113.281,Y -80.534,Z 250.000,A 0.000,B 0.000,C 180.000,E1 0.000} C_DIS
LIN {X 117.276,Y -74.597,Z 250.000,A 0.000,B 0.000,C 180.000,E1 0.000} C_DIS
LIN {X 120.961,Y -68.459,Z 250.000,A 0.000,B 0.000,C 180.000,E1 0.000} C_DIS
LIN {X 124.325,Y -62.141,Z 250.000,A 0.000,B 0.000,C 180.000,E1 0.000} C_DIS
LIN {X 127.360,Y -55.658,Z 250.000,A 0.000,B 0.000,C 180.000,E1 0.000} C_DIS
LIN {X 130.056,Y -49.029,Z 250.000,A 0.000,B 0.000,C 180.000,E1 0.000} C_DIS
LIN {X 132.407,Y -42.269,Z 250.000,A 0.000,B 0.000,C 180.000,E1 0.000} C_DIS
LIN {X 134.408,Y -35.397,Z 250.000,A 0.000,B 0.000,C 180.000,E1 0.000} C_DIS
LIN {X 136.051,Y -28.432,Z 250.000,A 0.000,B 0.000,C 180.000,E1 0.000} C_DIS
LIN {X 137.335,Y -21.390,Z 250.000,A 0.000,B 0.000,C 180.000,E1 0.000} C_DIS
LIN {X 138.254,Y -14.291,Z 250.000,A 0.000,B 0.000,C 180.000,E1 0.000} C_DIS
LIN {X 138.806,Y -7.155,Z 250.000,A 0.000,B 0.000,C 180.000,E1 0.000} C_DIS
LIN {X 138.990,Y 0.000,Z 250.000,A 0.000,B 0.000,C 180.000,E1 0.000} C_DIS
LIN {X 138.806,Y 7.155,Z 250.000,A 0.000,B 0.000,C 180.000,E1 0.000} C_DIS
LIN {X 138.254,Y 14.291,Z 250.000,A 0.000,B 0.000,C 180.000,E1 0.000} C_DIS
LIN {X 137.335,Y 21.390,Z 250.000,A 0.000,B 0.000,C 180.000,E1 0.000} C_DIS
LIN {X 136.051,Y 28.432,Z 250.000,A 0.000,B 0.000,C 180.000,E1 0.000} C_DIS
LIN {X 134.408,Y 35.397,Z 250.000,A 0.000,B 0.000,C 180.000,E1 0.000} C_DIS
LIN {X 132.407,Y 42.269,Z 250.000,A 0.000,B 0.000,C 180.000,E1 0.000} C_DIS
LIN {X 130.056,Y 49.029,Z 250.000,A 0.000,B 0.000,C 180.000,E1 0.000} C_DIS
LIN {X 127.360,Y 55.659,Z 250.000,A 0.000,B 0.000,C 180.000,E1 0.000} C_DIS
LIN {X 124.326,Y 62.140,Z 250.000,A 0.000,B 0.000,C 180.000,E1 0.000} C_DIS
LIN {X 120.961,Y 68.459,Z 250.000,A 0.000,B 0.000,C 180.000,E1 0.000} C_DIS
LIN {X 117.276,Y 74.597,Z 250.000,A 0.000,B 0.000,C 180.000,E1 0.000} C_DIS
LIN {X 113.281,Y 80.534,Z 250.000,A 0.000,B 0.000,C 180.000,E1 0.000} C_DIS
LIN {X 108.985,Y 86.258,Z 250.000,A 0.000,B 0.000,C 180.000,E1 0.000} C_DIS
LIN {X 104.400,Y 91.755,Z 250.000,A 0.000,B 0.000,C 180.000,E1 0.000} C_DIS
LIN {X 99.538,Y 97.008,Z 250.000,A 0.000,B 0.000,C 180.000,E1 0.000} C_DIS
LIN {X 94.413,Y 102.003,Z 250.000,A 0.000,B 0.000,C 180.000,E1 0.000} C_DIS
LIN {X 89.036,Y 106.728,Z 250.000,A 0.000,B 0.000,C 180.000,E1 0.000} C_DIS
LIN {X 83.424,Y 111.170,Z 250.000,A 0.000,B 0.000,C 180.000,E1 0.000} C_DIS
LIN {X 77.591,Y 115.317,Z 250.000,A 0.000,B 0.000,C 180.000,E1 0.000} C_DIS
LIN {X 71.551,Y 119.159,Z 250.000,A 0.000,B 0.000,C 180.000,E1 0.000} C_DIS
LIN {X 65.322,Y 122.684,Z 250.000,A 0.000,B 0.000,C 180.000,E1 0.000} C_DIS
LIN {X 58.920,Y 125.884,Z 250.000,A 0.000,B 0.000,C 180.000,E1 0.000} C_DIS
LIN {X 52.361,Y 128.751,Z 250.000,A 0.000,B 0.000,C 180.000,E1 0.000} C_DIS
LIN {X 45.667,Y 131.274,Z 250.000,A 0.000,B 0.000,C 180.000,E1 0.000} C_DIS
LIN {X 38.844,Y 133.451,Z 250.000,A 0.000,B 0.000,C 180.000,E1 0.000} C_DIS
LIN {X 31.922,Y 135.275,Z 250.000,A 0.000,B 0.000,C 180.000,E1 0.000} C_DIS
LIN {X 24.919,Y 136.739,Z 250.000,A 0.000,B 0.000,C 180.000,E1 0.000} C_DIS
LIN {X 17.847,Y 137.840,Z 250.000,A 0.000,B 0.000,C 180.000,E1 0.000} C_DIS
LIN {X 10.725,Y 138.576,Z 250.000,A 0.000,B 0.000,C 180.000,E1 0.000} C_DIS
LIN {X 3.577,Y 138.945,Z 250.000,A 0.000,B 0.000,C 180.000,E1 0.000} C_DIS
LIN {X -3.577,Y 138.945,Z 250.000,A 0.000,B 0.000,C 180.000,E1 0.000} C_DIS
LIN {X -10.725,Y 138.576,Z 250.000,A 0.000,B 0.000,C 180.000,E1 0.000} C_DIS
LIN {X -17.847,Y 137.840,Z 250.000,A 0.000,B 0.000,C 180.000,E1 0.000} C_DIS
LIN {X -24.920,Y 136.739,Z 250.000,A 0.000,B 0.000,C 180.000,E1 0.000} C_DIS
LIN {X -31.922,Y 135.275,Z 250.000,A 0.000,B 0.000,C 180.000,E1 0.000} C_DIS
LIN {X -38.844,Y 133.451,Z 250.000,A 0.000,B 0.000,C 180.000,E1 0.000} C_DIS
LIN {X -45.666,Y 131.274,Z 250.000,A 0.000,B 0.000,C 180.000,E1 0.000} C_DIS
LIN {X -52.362,Y 128.750,Z 250.000,A 0.000,B 0.000,C 180.000,E1 0.000} C_DIS
LIN {X -58.920,Y 125.884,Z 250.000,A 0.000,B 0.000,C 180.000,E1 0.000} C_DIS
LIN {X -65.322,Y 122.684,Z 250.000,A 0.000,B 0.000,C 180.000,E1 0.000} C_DIS
LIN {X -71.551,Y 119.159,Z 250.000,A 0.000,B 0.000,C 180.000,E1 0.000} C_DIS
LIN {X -77.591,Y 115.317,Z 250.000,A 0.000,B 0.000,C 180.000,E1 0.000} C_DIS
LIN {X -83.424,Y 111.170,Z 250.000,A 0.000,B 0.000,C 180.000,E1 0.000} C_DIS
LIN {X -89.036,Y 106.728,Z 250.000,A 0.000,B 0.000,C 180.000,E1 0.000} C_DIS
LIN {X -94.413,Y 102.003,Z 250.000,A 0.000,B 0.000,C 180.000,E1 0.000} C_DIS
LIN {X -99.538,Y 97.008,Z 250.000,A 0.000,B 0.000,C 180.000,E1 0.000} C_DIS
LIN {X -104.400,Y 91.755,Z 250.000,A 0.000,B 0.000,C 180.000,E1 0.000} C_DIS
LIN {X -108.985,Y 86.258,Z 250.000,A 0.000,B 0.000,C 180.000,E1 0.000} C_DIS
LIN {X -113.281,Y 80.534,Z 250.000,A 0.000,B 0.000,C 180.000,E1 0.000} C_DIS
LIN {X -117.276,Y 74.597,Z 250.000,A 0.000,B 0.000,C 180.000,E1 0.000} C_DIS
LIN {X -120.961,Y 68.459,Z 250.000,A 0.000,B 0.000,C 180.000,E1 0.000} C_DIS
LIN {X -124.325,Y 62.141,Z 250.000,A 0.000,B 0.000,C 180.000,E1 0.000} C_DIS
;rapid-leaky
$VEL.CP=0.3
LIN {X 68.537,Y -99.963,Z 250.000,A 0.000,B 0.000,C 180.000,E1 0.000} C_DIS
;bead-sparse_infill
$VEL.CP=0.32
LIN {X -99.954,Y 68.528,Z 250.000,A 0.000,B 0.000,C 180.000,E1 0.000} C_DIS
LIN {X -98.802,Y 70.240,Z 250.000,A 0.000,B 0.000,C 180.000,E1 0.000} C_DIS
LIN {X -95.055,Y 75.232,Z 250.000,A 0.000,B 0.000,C 180.000,E1 0.000} C_DIS
LIN {X -91.055,Y 80.027,Z 250.000,A 0.000,B 0.000,C 180.000,E1 0.000} C_DIS
LIN {X -86.815,Y 84.609,Z 250.000,A 0.000,B 0.000,C 180.000,E1 0.000} C_DIS
LIN {X -82.345,Y 88.965,Z 250.000,A 0.000,B 0.000,C 180.000,E1 0.000} C_DIS
LIN {X -77.656,Y 93.085,Z 250.000,A 0.000,B 0.000,C 180.000,E1 0.000} C_DIS
LIN {X -72.760,Y 96.961,Z 250.000,A 0.000,B 0.000,C 180.000,E1 0.000} C_DIS
LIN {X -67.673,Y 100.577,Z 250.000,A 0.000,B 0.000,C 180.000,E1 0.000} C_DIS
LIN {X -62.405,Y 103.928,Z 250.000,A 0.000,B 0.000,C 180.000,E1 0.000} C_DIS
LIN {X -56.973,Y 107.002,Z 250.000,A 0.000,B 0.000,C 180.000,E1 0.000} C_DIS
LIN {X -51.388,Y 109.794,Z 250.000,A 0.000,B 0.000,C 180.000,E1 0.000} C_DIS
LIN {X -45.670,Y 112.293,Z 250.000,A 0.000,B 0.000,C 180.000,E1 0.000} C_DIS
LIN {X -39.831,Y 114.494,Z 250.000,A 0.000,B 0.000,C 180.000,E1 0.000} C_DIS
LIN {X -33.879,Y 116.394,Z 250.000,A 0.000,B 0.000,C 180.000,E1 0.000} C_DIS
LIN {X -27.840,Y 117.985,Z 250.000,A 0.000,B 0.000,C 180.000,E1 0.000} C_DIS
LIN {X -21.735,Y 119.261,Z 250.000,A 0.000,B 0.000,C 180.000,E1 0.000} C_DIS
